LIN {X 0,Y 478.085,Z 266.813,A -85,B 0,C 180,E1 -7443.362,E2 -7443.362} C_VEL
LIN {X 0,Y 477.096,Z 286.447,A -85,B 0,C 180,E1 -7446.564,E2 -7446.564} C_VEL
LIN {X 0,Y 476.264,Z 303.664,A -85,B 0,C 180,E1 -7449.322,E2 -7449.322} C_VEL
LIN {X 0,Y 475.51,Z 306.267,A -85,B 0,C 180,E1 -7449.709,E2 -7449.709} C_VEL
LIN {X 0,Y 472.704,Z 310.776,A -85,B 0,C 180,E1 -7450.267,E2 -7450.267} C_VEL
LIN {X 0,Y 470.629,Z 314.949,A -85,B 0,C 180,E1 -7450.608,E2 -7450.608} C_VEL
LIN {X 0,Y 469.97,Z 318.585,A -85,B 0,C 180,E1 -7450.782,E2 -7450.782} C_VEL
LIN {X 0,Y 470.058,Z 319.87,A -85,B 0,C 180,E1 -7450.817,E2 -7450.817} C_VEL
LIN {X 0,Y 472.099,Z 332.179,A -85,B 0,C 180,E1 -7451.086,E2 -7451.086} C_VEL
LIN {X 0,Y 471.485,Z 425.613,A -85,B 0,C 180,E1 -7452.46,E2 -7452.46} C_VEL
LIN {X 0,Y 471.141,Z 438.708,A -85,B 0,C 180,E1 -7452.822,E2 -7452.822} C_VEL
LIN {X 0,Y 470.776,Z 451.277,A -85,B 0,C 180,E1 -7453.35,E2 -7453.35} C_VEL
LIN {X 0,Y 470.207,Z 463.7,A -85,B 0,C 180,E1 -7454.059,E2 -7454.059} C_VEL
LIN {X 0,Y 469.557,Z 475.266,A -85,B 0,C 180,E1 -7454.927,E2 -7454.927} C_VEL
LIN {X 0,Y 468.97,Z 485.65,A -85,B 0,C 180,E1 -7455.906,E2 -7455.906} C_VEL
LIN {X 0,Y 468.372,Z 495.014,A -85,B 0,C 180,E1 -7456.993,E2 -7456.993} C_VEL
LIN {X 0,Y 467.948,Z 502.687,A -85,B 0,C 180,E1 -7458.082,E2 -7458.082} C_VEL
LIN {X 0,Y 467.497,Z 510.197,A -85,B 0,C 180,E1 -7459.388,E2 -7459.388} C_VEL
LIN {X 0,Y 467.123,Z 517.124,A -85,B 0,C 180,E1 -7460.911,E2 -7460.911} C_VEL
LIN {X 0,Y 466.94,Z 521.744,A -85,B 0,C 180,E1 -7462.215,E2 -7462.215} C_VEL
LIN {X 0,Y 466.794,Z 525.41,A -85,B 0,C 180,E1 -7463.564,E2 -7463.564} C_VEL
LIN {X 0,Y 466.711,Z 527.879,A -85,B 0,C 180,E1 -7464.816,E2 -7464.816} C_VEL
LIN {X 0,Y 466.716,Z 529.948,A -85,B 0,C 180,E1 -7466.547,E2 -7466.547} C_VEL
LIN {X 0,Y 466.632,Z 530.463,A -85,B 0,C 180,E1 -7468.274,E2 -7468.274} C_VEL
LIN {X 0,Y 466.604,Z 529.509,A -85,B 0,C 180,E1 -7470,E2 -7470} C_VEL
LIN {X 0,Y 466.628,Z 528.478,A -85,B 0,C 180,E1 -7470.863,E2 -7470.863} C_VEL
LIN {X 0,Y 466.719,Z 527.02,A -85,B 0,C 180,E1 -7471.726,E2 -7471.726} C_VEL
LIN {X 0,Y 466.936,Z 522.899,A -85,B 0,C 180,E1 -7473.451,E2 -7473.451} C_VEL
LIN {X 0,Y 467.13,Z 518.624,A -85,B 0,C 180,E1 -7474.746,E2 -7474.746} C_VEL
LIN {X 0,Y 467.264,Z 513.213,A -85,B 0,C 180,E1 -7476.043,E2 -7476.043} C_VEL
LIN {X 0,Y 467.751,Z 506.1,A -85,B 0,C 180,E1 -7477.402,E2 -7477.402} C_VEL
LIN {X 0,Y 468.164,Z 498.071,A -85,B 0,C 180,E1 -7478.634,E2 -7478.634} C_VEL
LIN {X 0,Y 468.673,Z 489.478,A -85,B 0,C 180,E1 -7479.712,E2 -7479.712} C_VEL
LIN {X 0,Y 469.27,Z 478.914,A -85,B 0,C 180,E1 -7480.79,E2 -7480.79} C_VEL
LIN {X 0,Y 469.812,Z 468.39,A -85,B 0,C 180,E1 -7481.651,E2 -7481.651} C_VEL
LIN {X 0,Y 470.413,Z 456.63,A -85,B 0,C 180,E1 -7482.401,E2 -7482.401} C_VEL
LIN {X 0,Y 470.831,Z 444.4,A -85,B 0,C 180,E1 -7482.993,E2 -7482.993} C_VEL
LIN {X 0,Y 471.2,Z 431.794,A -85,B 0,C 180,E1 -7483.421,E2 -7483.421} C_VEL
LIN {X 0,Y 471.404,Z 418.703,A -85,B 0,C 180,E1 -7483.69,E2 -7483.69} C_VEL
LIN {X 0,Y 471.889,Z 331.972,A -85,B 0,C 180,E1 -7484.942,E2 -7484.942} C_VEL
LIN {X 0,Y 468.922,Z 314.095,A -85,B 0,C 180,E1 -7485.344,E2 -7485.344} C_VEL
LIN {X 0,Y 469.676,Z 295.344,A -85,B 0,C 180,E1 -7488.314,E2 -7488.314} C_VEL
LIN {X 0,Y 470.606,Z 276.031,A -85,B 0,C 180,E1 -7491.461,E2 -7491.461} C_VEL
LIN {X 0,Y 471.155,Z 266.374,A -85,B 0,C 180,E1 -7493.051,E2 -7493.051} C_VEL
LIN {X 0,Y 468.554,Z 254.185,A -85,B 0,C 180,E1 -7495.274,E2 -7495.274} C_VEL
LIN {X 0,Y 467.634,Z 249.988,A -85,B 0,C 180,E1 -7496.077,E2 -7496.077} C_VEL
LIN {X 0,Y 467.579,Z 249.864,A -85,B 0,C 180,E1 -7498.749,E2 -7498.749} C_VEL
LIN {X 0,Y 467.585,Z 249.866,A -85,B 0,C 180,E1 -7501.739,E2 -7501.739} C_VEL
LIN {X 0,Y 467.565,Z 249.859,A -85,B 0,C 180,E1 -7504.832,E2 -7504.832} C_VEL
LIN {X 0,Y 467.565,Z 249.864,A -85,B 0,C 180,E1 -7508.044,E2 -7508.044} C_VEL
LIN {X 0,Y 467.582,Z 249.863,A -85,B 0,C 180,E1 -7511.276,E2 -7511.276} C_VEL
LIN {X 0,Y 467.566,Z 249.864,A -85,B 0,C 180,E1 -7513.822,E2 -7513.822} C_VEL
LIN {X 0,Y 467.554,Z 249.863,A -85,B 0,C 180,E1 -7516.255,E2 -7516.255} C_VEL
LIN {X 0,Y 467.576,Z 249.866,A -85,B 0,C 180,E1 -7518.722,E2 -7518.722} C_VEL
LIN {X 0,Y 467.563,Z 249.864,A -85,B 0,C 180,E1 -7521.955,E2 -7521.955} C_VEL
LIN {X 0,Y 467.565,Z 249.858,A -85,B 0,C 180,E1 -7525.167,E2 -7525.167} C_VEL
LIN {X 0,Y 467.582,Z 249.859,A -85,B 0,C 180,E1 -7528.259,E2 -7528.259} C_VEL
LIN {X 0,Y 467.578,Z 249.863,A -85,B 0,C 180,E1 -7531.25,E2 -7531.25} C_VEL
LIN {X 0,Y 467.605,Z 249.86,A -85,B 0,C 180,E1 -7534.159,E2 -7534.159} C_VEL
LIN {X 0,Y 467.572,Z 249.87,A -85,B 0,C 180,E1 -7536.995,E2 -7536.995} C_VEL
LIN {X 0,Y 467.617,Z 249.854,A -85,B 0,C 180,E1 -7539.777,E2 -7539.777} C_VEL
LIN {X 0,Y 467.604,Z 249.863,A -85,B 0,C 180,E1 -7542.506,E2 -7542.506} C_VEL
LIN {X 0,Y 467.601,Z 249.859,A -85,B 0,C 180,E1 -7545.196,E2 -7545.196} C_VEL
LIN {X 0,Y 467.649,Z 249.854,A -85,B 0,C 180,E1 -7547.854,E2 -7547.854} C_VEL
LIN {X 0,Y 467.675,Z 249.85,A -85,B 0,C 180,E1 -7551.357,E2 -7551.357} C_VEL
LIN {X 0,Y 467.737,Z 249.844,A -85,B 0,C 180,E1 -7553.962,E2 -7553.962} C_VEL
LIN {X 0,Y 467.853,Z 249.828,A -85,B 0,C 180,E1 -7557.417,E2 -7557.417} C_VEL
LIN {X 0,Y 467.875,Z 249.826,A -85,B 0,C 180,E1 -7560,E2 -7560} C_VEL
LIN {X 0,Y 467.853,Z 249.834,A -85,B 0,C 180,E1 -7562.583,E2 -7562.583} C_VEL
LIN {X 0,Y 467.736,Z 249.842,A -85,B 0,C 180,E1 -7566.037,E2 -7566.037} C_VEL
LIN {X 0,Y 467.674,Z 249.854,A -85,B 0,C 180,E1 -7568.643,E2 -7568.643} C_VEL
LIN {X 0,Y 467.648,Z 249.855,A -85,B 0,C 180,E1 -7572.145,E2 -7572.145} C_VEL
LIN {X 0,Y 467.632,Z 249.855,A -85,B 0,C 180,E1 -7575.695,E2 -7575.695} C_VEL
LIN {X 0,Y 467.61,Z 249.859,A -85,B 0,C 180,E1 -7578.765,E2 -7578.765} C_VEL
LIN {X 0,Y 467.573,Z 249.861,A -85,B 0,C 180,E1 -7581.268,E2 -7581.268} C_VEL
LIN {X 0,Y 467.567,Z 249.869,A -85,B 0,C 180,E1 -7583.943,E2 -7583.943} C_VEL
LIN {X 0,Y 467.61,Z 249.859,A -85,B 0,C 180,E1 -7586.801,E2 -7586.801} C_VEL
LIN {X 0,Y 467.581,Z 249.856,A -85,B 0,C 180,E1 -7589.736,E2 -7589.736} C_VEL
LIN {X 0,Y 467.578,Z 249.863,A -85,B 0,C 180,E1 -7592.759,E2 -7592.759} C_VEL
LIN {X 0,Y 467.551,Z 249.863,A -85,B 0,C 180,E1 -7595.89,E2 -7595.89} C_VEL
LIN {X 0,Y 467.577,Z 249.864,A -85,B 0,C 180,E1 -7599.145,E2 -7599.145} C_VEL
LIN {X 0,Y 467.582,Z 249.859,A -85,B 0,C 180,E1 -7602.567,E2 -7602.567} C_VEL
LIN {X 0,Y 467.566,Z 249.866,A -85,B 0,C 180,E1 -7605.054,E2 -7605.054} C_VEL
LIN {X 0,Y 467.585,Z 249.844,A -85,B 0,C 180,E1 -7607.44,E2 -7607.44} C_VEL
LIN {X 0,Y 467.578,Z 249.863,A -85,B 0,C 180,E1 -7610.856,E2 -7610.856} C_VEL
LIN {X 0,Y 467.557,Z 249.852,A -85,B 0,C 180,E1 -7614.261,E2 -7614.261} C_VEL
LIN {X 0,Y 467.58,Z 249.861,A -85,B 0,C 180,E1 -7617.321,E2 -7617.321} C_VEL
LIN {X 0,Y 467.568,Z 249.865,A -85,B 0,C 180,E1 -7620.668,E2 -7620.668} C_VEL
LIN {X 0,Y 467.679,Z 249.999,A -85,B 0,C 180,E1 -7622.625,E2 -7622.625} C_VEL
LIN {X 0,Y 471.47,Z 266.255,A -85,B 0,C 180,E1 -7625.331,E2 -7625.331} C_VEL
LIN {X 0,Y 471.671,Z 269.572,A -85,B 0,C 180,E1 -7625.836,E2 -7625.836} C_VEL
LIN {X 0,Y 470.357,Z 291.394,A -85,B 0,C 180,E1 -7628.986,E2 -7628.986} C_VEL
LIN {X 0,Y 470.145,Z 296.887,A -85,B 0,C 180,E1 -7629.737,E2 -7629.737} C_VEL
LIN {X 0,Y 472.697,Z 313.021,A -85,B 0,C 180,E1 -7630.12,E2 -7630.12} C_VEL
LIN {X 0,Y 471.417,Z 431.926,A -85,B 0,C 180,E1 -7632.037,E2 -7632.037} C_VEL
LIN {X 0,Y 471.033,Z 446.54,A -85,B 0,C 180,E1 -7632.442,E2 -7632.442} C_VEL
LIN {X 0,Y 470.559,Z 460.601,A -85,B 0,C 180,E1 -7633.016,E2 -7633.016} C_VEL
LIN {X 0,Y 470.028,Z 473.558,A -85,B 0,C 180,E1 -7633.719,E2 -7633.719} C_VEL
LIN {X 0,Y 469.39,Z 486.203,A -85,B 0,C 180,E1 -7634.588,E2 -7634.588} C_VEL
LIN {X 0,Y 468.797,Z 497.744,A -85,B 0,C 180,E1 -7635.568,E2 -7635.568} C_VEL
LIN {X 0,Y 468.358,Z 507.345,A -85,B 0,C 180,E1 -7636.551,E2 -7636.551} C_VEL
LIN {X 0,Y 467.91,Z 518.036,A -85,B 0,C 180,E1 -7637.862,E2 -7637.862} C_VEL
LIN {X 0,Y 467.454,Z 526.834,A -85,B 0,C 180,E1 -7639.168,E2 -7639.168} C_VEL
LIN {X 0,Y 467.105,Z 535.228,A -85,B 0,C 180,E1 -7640.692,E2 -7640.692} C_VEL
LIN {X 0,Y 466.851,Z 541.954,A -85,B 0,C 180,E1 -7642.213,E2 -7642.213} C_VEL
LIN {X 0,Y 466.757,Z 546.875,A -85,B 0,C 180,E1 -7643.6,E2 -7643.6} C_VEL
LIN {X 0,Y 466.723,Z 550.262,A -85,B 0,C 180,E1 -7644.816,E2 -7644.816} C_VEL
LIN {X 0,Y 466.679,Z 553.826,A -85,B 0,C 180,E1 -7646.547,E2 -7646.547} C_VEL
LIN {X 0,Y 466.604,Z 555.941,A -85,B 0,C 180,E1 -7648.274,E2 -7648.274} C_VEL
LIN {X 0,Y 466.597,Z 556.653,A -85,B 0,C 180,E1 -7650,E2 -7650} C_VEL
LIN {X 0,Y 466.604,Z 555.958,A -85,B 0,C 180,E1 -7651.726,E2 -7651.726} C_VEL
LIN {X 0,Y 466.679,Z 553.86,A -85,B 0,C 180,E1 -7653.453,E2 -7653.453} C_VEL
LIN {X 0,Y 466.727,Z 550.313,A -85,B 0,C 180,E1 -7655.184,E2 -7655.184} C_VEL
LIN {X 0,Y 466.82,Z 545.216,A -85,B 0,C 180,E1 -7656.917,E2 -7656.917} C_VEL
LIN {X 0,Y 466.947,Z 540.274,A -85,B 0,C 180,E1 -7658.22,E2 -7658.22} C_VEL
LIN {X 0,Y 467.177,Z 533.133,A -85,B 0,C 180,E1 -7659.743,E2 -7659.743} C_VEL
LIN {X 0,Y 467.617,Z 524.274,A -85,B 0,C 180,E1 -7661.267,E2 -7661.267} C_VEL
LIN {X 0,Y 468.088,Z 514.113,A -85,B 0,C 180,E1 -7662.69,E2 -7662.69} C_VEL
LIN {X 0,Y 468.575,Z 503.701,A -85,B 0,C 180,E1 -7663.885,E2 -7663.885} C_VEL
LIN {X 0,Y 469.161,Z 492.153,A -85,B 0,C 180,E1 -7664.975,E2 -7664.975} C_VEL
LIN {X 0,Y 469.84,Z 479.364,A -85,B 0,C 180,E1 -7665.953,E2 -7665.953} C_VEL
LIN {X 0,Y 470.412,Z 465.977,A -85,B 0,C 180,E1 -7666.766,E2 -7666.766} C_VEL
LIN {X 0,Y 470.96,Z 451.819,A -85,B 0,C 180,E1 -7667.42,E2 -7667.42} C_VEL
LIN {X 0,Y 471.441,Z 437.698,A -85,B 0,C 180,E1 -7667.878,E2 -7667.878} C_VEL
LIN {X 0,Y 471.723,Z 421.368,A -85,B 0,C 180,E1 -7668.204,E2 -7668.204} C_VEL
LIN {X 0,Y 472.823,Z 312.677,A -85,B 0,C 180,E1 -7669.954,E2 -7669.954} C_VEL
LIN {X 0,Y 470.225,Z 296.843,A -85,B 0,C 180,E1 -7670.346,E2 -7670.346} C_VEL
LIN {X 0,Y 471.398,Z 276.465,A -85,B 0,C 180,E1 -7673.271,E2 -7673.271} C_VEL
LIN {X 0,Y 471.885,Z 268.33,A -85,B 0,C 180,E1 -7674.461,E2 -7674.461} C_VEL
LIN {X 0,Y 468.859,Z 254.709,A -85,B 0,C 180,E1 -7676.723,E2 -7676.723} C_VEL
LIN {X 0,Y 467.644,Z 249.964,A -85,B 0,C 180,E1 -7677.581,E2 -7677.581} C_VEL
LIN {X 0,Y 467.567,Z 249.86,A -85,B 0,C 180,E1 -7681.045,E2 -7681.045} C_VEL
LIN {X 0,Y 467.586,Z 249.869,A -85,B 0,C 180,E1 -7684.242,E2 -7684.242} C_VEL
LIN {X 0,Y 467.545,Z 249.857,A -85,B 0,C 180,E1 -7687.186,E2 -7687.186} C_VEL
LIN {X 0,Y 467.575,Z 249.865,A -85,B 0,C 180,E1 -7690.264,E2 -7690.264} C_VEL
LIN {X 0,Y 467.616,Z 249.863,A -85,B 0,C 180,E1 -7692.571,E2 -7692.571} C_VEL
LIN {X 0,Y 467.567,Z 249.862,A -85,B 0,C 180,E1 -7695.053,E2 -7695.053} C_VEL
LIN {X 0,Y 467.585,Z 249.862,A -85,B 0,C 180,E1 -7697.44,E2 -7697.44} C_VEL
LIN {X 0,Y 467.578,Z 249.865,A -85,B 0,C 180,E1 -7700.855,E2 -7700.855} C_VEL
LIN {X 0,Y 467.558,Z 249.86,A -85,B 0,C 180,E1 -7704.26,E2 -7704.26} C_VEL
LIN {X 0,Y 467.577,Z 249.864,A -85,B 0,C 180,E1 -7707.32,E2 -7707.32} C_VEL
LIN {X 0,Y 467.571,Z 249.855,A -85,B 0,C 180,E1 -7710.666,E2 -7710.666} C_VEL
LIN {X 0,Y 467.61,Z 249.859,A -85,B 0,C 180,E1 -7713.199,E2 -7713.199} C_VEL
LIN {X 0,Y 467.587,Z 249.863,A -85,B 0,C 180,E1 -7716.468,E2 -7716.468} C_VEL
LIN {X 0,Y 467.616,Z 249.86,A -85,B 0,C 180,E1 -7719.777,E2 -7719.777} C_VEL
LIN {X 0,Y 467.603,Z 249.859,A -85,B 0,C 180,E1 -7722.507,E2 -7722.507} C_VEL
LIN {X 0,Y 467.6,Z 249.86,A -85,B 0,C 180,E1 -7725.196,E2 -7725.196} C_VEL
LIN {X 0,Y 467.649,Z 249.854,A -85,B 0,C 180,E1 -7727.855,E2 -7727.855} C_VEL
LIN {X 0,Y 467.675,Z 249.854,A -85,B 0,C 180,E1 -7731.357,E2 -7731.357} C_VEL
LIN {X 0,Y 467.737,Z 249.847,A -85,B 0,C 180,E1 -7733.963,E2 -7733.963} C_VEL
LIN {X 0,Y 467.853,Z 249.83,A -85,B 0,C 180,E1 -7737.417,E2 -7737.417} C_VEL
LIN {X 0,Y 467.876,Z 249.828,A -85,B 0,C 180,E1 -7740,E2 -7740} C_VEL
LIN {X 0,Y 467.854,Z 249.823,A -85,B 0,C 180,E1 -7742.583,E2 -7742.583} C_VEL
LIN {X 0,Y 467.737,Z 249.841,A -85,B 0,C 180,E1 -7746.038,E2 -7746.038} C_VEL
LIN {X 0,Y 467.676,Z 249.85,A -85,B 0,C 180,E1 -7748.643,E2 -7748.643} C_VEL
LIN {X 0,Y 467.65,Z 249.852,A -85,B 0,C 180,E1 -7752.146,E2 -7752.146} C_VEL
LIN {X 0,Y 467.633,Z 249.855,A -85,B 0,C 180,E1 -7755.696,E2 -7755.696} C_VEL
LIN {X 0,Y 467.612,Z 249.861,A -85,B 0,C 180,E1 -7758.765,E2 -7758.765} C_VEL
LIN {X 0,Y 467.576,Z 249.869,A -85,B 0,C 180,E1 -7761.269,E2 -7761.269} C_VEL
LIN {X 0,Y 467.568,Z 249.862,A -85,B 0,C 180,E1 -7763.944,E2 -7763.944} C_VEL
LIN {X 0,Y 467.613,Z 249.863,A -85,B 0,C 180,E1 -7766.801,E2 -7766.801} C_VEL
LIN {X 0,Y 467.55,Z 249.861,A -85,B 0,C 180,E1 -7769.739,E2 -7769.739} C_VEL
LIN {X 0,Y 467.581,Z 249.868,A -85,B 0,C 180,E1 -7772.759,E2 -7772.759} C_VEL
LIN {X 0,Y 467.554,Z 249.861,A -85,B 0,C 180,E1 -7775.89,E2 -7775.89} C_VEL
LIN {X 0,Y 467.574,Z 249.86,A -85,B 0,C 180,E1 -7779.146,E2 -7779.146} C_VEL
LIN {X 0,Y 467.585,Z 249.867,A -85,B 0,C 180,E1 -7782.568,E2 -7782.568} C_VEL
LIN {X 0,Y 467.57,Z 249.868,A -85,B 0,C 180,E1 -7785.054,E2 -7785.054} C_VEL
LIN {X 0,Y 467.589,Z 249.859,A -85,B 0,C 180,E1 -7787.441,E2 -7787.441} C_VEL
LIN {X 0,Y 467.582,Z 249.851,A -85,B 0,C 180,E1 -7790.856,E2 -7790.856} C_VEL
LIN {X 0,Y 467.56,Z 249.871,A -85,B 0,C 180,E1 -7794.262,E2 -7794.262} C_VEL
LIN {X 0,Y 467.581,Z 249.867,A -85,B 0,C 180,E1 -7797.322,E2 -7797.322} C_VEL
LIN {X 0,Y 467.596,Z 250.065,A -85,B 0,C 180,E1 -7799.831,E2 -7799.831} C_VEL
LIN {X 0,Y 470.568,Z 262.803,A -85,B 0,C 180,E1 -7802.246,E2 -7802.246} C_VEL
LIN {X 0,Y 471.257,Z 268.059,A -85,B 0,C 180,E1 -7803.184,E2 -7803.184} C_VEL
LIN {X 0,Y 470.191,Z 287.705,A -85,B 0,C 180,E1 -7806.433,E2 -7806.433} C_VEL
LIN {X 0,Y 469.158,Z 308.757,A -85,B 0,C 180,E1 -7809.847,E2 -7809.847} C_VEL
LIN {X 0,Y 469.023,Z 313.903,A -85,B 0,C 180,E1 -7810.648,E2 -7810.648} C_VEL
LIN {X 0,Y 470.058,Z 319.87,A -85,B 0,C 180,E1 -7810.817,E2 -7810.817} C_VEL
LIN {X 0,Y 470.179,Z 325.726,A -85,B 0,C 180,E1 -7810.91,E2 -7810.91} C_VEL
LIN {X 0,Y 469.247,Z 331.594,A -85,B 0,C 180,E1 -7810.958,E2 -7810.958} C_VEL
LIN {X 0,Y 466.333,Z 343.281,A -85,B 0,C 180,E1 -7811.009,E2 -7811.009} C_VEL
LIN {X 0,Y 465.398,Z 349.209,A -85,B 0,C 180,E1 -7811.058,E2 -7811.058} C_VEL
LIN {X 0,Y 465.298,Z 351.201,A -85,B 0,C 180,E1 -7811.084,E2 -7811.084} C_VEL
LIN {X 0,Y 464.726,Z 425.765,A -85,B 0,C 180,E1 -7812.196,E2 -7812.196} C_VEL
LIN {X 0,Y 464.36,Z 439.005,A -85,B 0,C 180,E1 -7812.569,E2 -7812.569} C_VEL
LIN {X 0,Y 463.967,Z 451.581,A -85,B 0,C 180,E1 -7813.107,E2 -7813.107} C_VEL
LIN {X 0,Y 463.395,Z 463.826,A -85,B 0,C 180,E1 -7813.819,E2 -7813.819} C_VEL
LIN {X 0,Y 462.694,Z 475.393,A -85,B 0,C 180,E1 -7814.698,E2 -7814.698} C_VEL
LIN {X 0,Y 462.066,Z 485.78,A -85,B 0,C 180,E1 -7815.691,E2 -7815.691} C_VEL
LIN {X 0,Y 461.419,Z 495.148,A -85,B 0,C 180,E1 -7816.793,E2 -7816.793} C_VEL
LIN {X 0,Y 460.977,Z 502.825,A -85,B 0,C 180,E1 -7817.899,E2 -7817.899} C_VEL
LIN {X 0,Y 460.498,Z 510.341,A -85,B 0,C 180,E1 -7819.225,E2 -7819.225} C_VEL
LIN {X 0,Y 460.093,Z 517.272,A -85,B 0,C 180,E1 -7820.771,E2 -7820.771} C_VEL
LIN {X 0,Y 459.886,Z 521.898,A -85,B 0,C 180,E1 -7822.095,E2 -7822.095} C_VEL
LIN {X 0,Y 459.717,Z 525.817,A -85,B 0,C 180,E1 -7823.569,E2 -7823.569} C_VEL
LIN {X 0,Y 459.646,Z 528.049,A -85,B 0,C 180,E1 -7824.736,E2 -7824.736} C_VEL
LIN {X 0,Y 459.613,Z 530.13,A -85,B 0,C 180,E1 -7826.493,E2 -7826.493} C_VEL
LIN {X 0,Y 459.585,Z 530.591,A -85,B 0,C 180,E1 -7827.371,E2 -7827.371} C_VEL
LIN {X 0,Y 459.525,Z 530.378,A -85,B 0,C 180,E1 -7829.124,E2 -7829.124} C_VEL
LIN {X 0,Y 459.562,Z 528.711,A -85,B 0,C 180,E1 -7830.876,E2 -7830.876} C_VEL
LIN {X 0,Y 459.627,Z 527.272,A -85,B 0,C 180,E1 -7831.752,E2 -7831.752} C_VEL
LIN {X 0,Y 459.867,Z 523.177,A -85,B 0,C 180,E1 -7833.505,E2 -7833.505} C_VEL
LIN {X 0,Y 460.069,Z 518.929,A -85,B 0,C 180,E1 -7834.819,E2 -7834.819} C_VEL
LIN {X 0,Y 460.291,Z 512.552,A -85,B 0,C 180,E1 -7836.355,E2 -7836.355} C_VEL
LIN {X 0,Y 460.777,Z 505.573,A -85,B 0,C 180,E1 -7837.669,E2 -7837.669} C_VEL
LIN {X 0,Y 461.172,Z 498.514,A -85,B 0,C 180,E1 -7838.765,E2 -7838.765} C_VEL
LIN {X 0,Y 461.703,Z 489.98,A -85,B 0,C 180,E1 -7839.86,E2 -7839.86} C_VEL
LIN {X 0,Y 462.332,Z 479.485,A -85,B 0,C 180,E1 -7840.953,E2 -7840.953} C_VEL
LIN {X 0,Y 462.909,Z 469.056,A -85,B 0,C 180,E1 -7841.827,E2 -7841.827} C_VEL
LIN {X 0,Y 463.545,Z 457.506,A -85,B 0,C 180,E1 -7842.588,E2 -7842.588} C_VEL
LIN {X 0,Y 463.965,Z 445.517,A -85,B 0,C 180,E1 -7843.189,E2 -7843.189} C_VEL
LIN {X 0,Y 464.384,Z 432.407,A -85,B 0,C 180,E1 -7843.65,E2 -7843.65} C_VEL
LIN {X 0,Y 464.611,Z 419.813,A -85,B 0,C 180,E1 -7843.922,E2 -7843.922} C_VEL
LIN {X 0,Y 465.011,Z 331.821,A -85,B 0,C 180,E1 -7845.213,E2 -7845.213} C_VEL
LIN {X 0,Y 462.025,Z 314.35,A -85,B 0,C 180,E1 -7845.607,E2 -7845.607} C_VEL
LIN {X 0,Y 461.99,Z 313.56,A -85,B 0,C 180,E1 -7845.665,E2 -7845.665} C_VEL
LIN {X 0,Y 462.925,Z 292.706,A -85,B 0,C 180,E1 -7849.05,E2 -7849.05} C_VEL
LIN {X 0,Y 463.914,Z 273.38,A -85,B 0,C 180,E1 -7852.255,E2 -7852.255} C_VEL
LIN {X 0,Y 464.285,Z 267.857,A -85,B 0,C 180,E1 -7853.176,E2 -7853.176} C_VEL
LIN {X 0,Y 461.309,Z 254.051,A -85,B 0,C 180,E1 -7855.741,E2 -7855.741} C_VEL
LIN {X 0,Y 460.582,Z 250.828,A -85,B 0,C 180,E1 -7856.385,E2 -7856.385} C_VEL
LIN {X 0,Y 460.542,Z 250.734,A -85,B 0,C 180,E1 -7859.23,E2 -7859.23} C_VEL
LIN {X 0,Y 460.533,Z 250.741,A -85,B 0,C 180,E1 -7862.284,E2 -7862.284} C_VEL
LIN {X 0,Y 460.511,Z 250.745,A -85,B 0,C 180,E1 -7865.445,E2 -7865.445} C_VEL
LIN {X 0,Y 460.544,Z 250.741,A -85,B 0,C 180,E1 -7868.897,E2 -7868.897} C_VEL
LIN {X 0,Y 460.523,Z 250.742,A -85,B 0,C 180,E1 -7872.18,E2 -7872.18} C_VEL
LIN {X 0,Y 460.516,Z 250.741,A -85,B 0,C 180,E1 -7875.411,E2 -7875.411} C_VEL
LIN {X 0,Y 460.53,Z 250.741,A -85,B 0,C 180,E1 -7878.397,E2 -7878.397} C_VEL
LIN {X 0,Y 460.517,Z 250.741,A -85,B 0,C 180,E1 -7881.265,E2 -7881.265} C_VEL
LIN {X 0,Y 460.51,Z 250.744,A -85,B 0,C 180,E1 -7884.554,E2 -7884.554} C_VEL
LIN {X 0,Y 460.529,Z 250.737,A -85,B 0,C 180,E1 -7887.715,E2 -7887.715} C_VEL
LIN {X 0,Y 460.543,Z 250.745,A -85,B 0,C 180,E1 -7890.769,E2 -7890.769} C_VEL
LIN {X 0,Y 460.558,Z 250.738,A -85,B 0,C 180,E1 -7893.734,E2 -7893.734} C_VEL
LIN {X 0,Y 460.541,Z 250.739,A -85,B 0,C 180,E1 -7896.623,E2 -7896.623} C_VEL
LIN {X 0,Y 460.545,Z 250.736,A -85,B 0,C 180,E1 -7899.452,E2 -7899.452} C_VEL
LIN {X 0,Y 460.554,Z 250.739,A -85,B 0,C 180,E1 -7902.23,E2 -7902.23} C_VEL
LIN {X 0,Y 460.559,Z 250.737,A -85,B 0,C 180,E1 -7904.964,E2 -7904.964} C_VEL
LIN {X 0,Y 460.602,Z 250.732,A -85,B 0,C 180,E1 -7907.665,E2 -7907.665} C_VEL
LIN {X 0,Y 460.622,Z 250.729,A -85,B 0,C 180,E1 -7911.223,E2 -7911.223} C_VEL
LIN {X 0,Y 460.703,Z 250.719,A -85,B 0,C 180,E1 -7913.87,E2 -7913.87} C_VEL
LIN {X 0,Y 460.818,Z 250.705,A -85,B 0,C 180,E1 -7917.377,E2 -7917.377} C_VEL
LIN {X 0,Y 460.846,Z 250.702,A -85,B 0,C 180,E1 -7920,E2 -7920} C_VEL
LIN {X 0,Y 460.818,Z 250.71,A -85,B 0,C 180,E1 -7922.622,E2 -7922.622} C_VEL
LIN {X 0,Y 460.703,Z 250.718,A -85,B 0,C 180,E1 -7926.13,E2 -7926.13} C_VEL
LIN {X 0,Y 460.622,Z 250.731,A -85,B 0,C 180,E1 -7928.776,E2 -7928.776} C_VEL
LIN {X 0,Y 460.606,Z 250.737,A -85,B 0,C 180,E1 -7932.445,E2 -7932.445} C_VEL
LIN {X 0,Y 460.593,Z 250.733,A -85,B 0,C 180,E1 -7935.998,E2 -7935.998} C_VEL
LIN {X 0,Y 460.563,Z 250.736,A -85,B 0,C 180,E1 -7938.902,E2 -7938.902} C_VEL
LIN {X 0,Y 460.509,Z 250.742,A -85,B 0,C 180,E1 -7941.486,E2 -7941.486} C_VEL
LIN {X 0,Y 460.536,Z 250.74,A -85,B 0,C 180,E1 -7944.332,E2 -7944.332} C_VEL
LIN {X 0,Y 460.573,Z 250.736,A -85,B 0,C 180,E1 -7947.244,E2 -7947.244} C_VEL
LIN {X 0,Y 460.521,Z 250.731,A -85,B 0,C 180,E1 -7950.239,E2 -7950.239} C_VEL
LIN {X 0,Y 460.524,Z 250.743,A -85,B 0,C 180,E1 -7953.325,E2 -7953.325} C_VEL
LIN {X 0,Y 460.473,Z 250.737,A -85,B 0,C 180,E1 -7956.53,E2 -7956.53} C_VEL
LIN {X 0,Y 460.553,Z 250.745,A -85,B 0,C 180,E1 -7959.86,E2 -7959.86} C_VEL
LIN {X 0,Y 460.508,Z 250.74,A -85,B 0,C 180,E1 -7962.901,E2 -7962.901} C_VEL
LIN {X 0,Y 460.505,Z 250.74,A -85,B 0,C 180,E1 -7965.831,E2 -7965.831} C_VEL
LIN {X 0,Y 460.527,Z 250.722,A -85,B 0,C 180,E1 -7968.989,E2 -7968.989} C_VEL
LIN {X 0,Y 460.522,Z 250.746,A -85,B 0,C 180,E1 -7971.267,E2 -7971.267} C_VEL
LIN {X 0,Y 460.507,Z 250.73,A -85,B 0,C 180,E1 -7974.555,E2 -7974.555} C_VEL
LIN {X 0,Y 460.529,Z 250.733,A -85,B 0,C 180,E1 -7977.716,E2 -7977.716} C_VEL
LIN {X 0,Y 460.538,Z 250.738,A -85,B 0,C 180,E1 -7980.77,E2 -7980.77} C_VEL
LIN {X 0,Y 460.646,Z 250.959,A -85,B 0,C 180,E1 -7982.341,E2 -7982.341} C_VEL
LIN {X 0,Y 464.19,Z 266.18,A -85,B 0,C 180,E1 -7984.918,E2 -7984.918} C_VEL
LIN {X 0,Y 464.86,Z 270.105,A -85,B 0,C 180,E1 -7985.55,E2 -7985.55} C_VEL
LIN {X 0,Y 463.651,Z 289.726,A -85,B 0,C 180,E1 -7988.434,E2 -7988.434} C_VEL
LIN {X 0,Y 463.272,Z 297.079,A -85,B 0,C 180,E1 -7989.461,E2 -7989.461} C_VEL
LIN {X 0,Y 465.969,Z 313.961,A -85,B 0,C 180,E1 -7989.869,E2 -7989.869} C_VEL
LIN {X 0,Y 464.586,Z 432.822,A -85,B 0,C 180,E1 -7991.82,E2 -7991.82} C_VEL
LIN {X 0,Y 464.162,Z 447.086,A -85,B 0,C 180,E1 -7992.231,E2 -7992.231} C_VEL
LIN {X 0,Y 463.666,Z 460.989,A -85,B 0,C 180,E1 -7992.813,E2 -7992.813} C_VEL
LIN {X 0,Y 463.095,Z 474.719,A -85,B 0,C 180,E1 -7993.582,E2 -7993.582} C_VEL
LIN {X 0,Y 462.414,Z 487.118,A -85,B 0,C 180,E1 -7994.463,E2 -7994.463} C_VEL
LIN {X 0,Y 461.792,Z 498.474,A -85,B 0,C 180,E1 -7995.457,E2 -7995.457} C_VEL
LIN {X 0,Y 461.295,Z 508.92,A -85,B 0,C 180,E1 -7996.565,E2 -7996.565} C_VEL
LIN {X 0,Y 460.816,Z 519.265,A -85,B 0,C 180,E1 -7997.895,E2 -7997.895} C_VEL
LIN {X 0,Y 460.371,Z 527.818,A -85,B 0,C 180,E1 -7999.222,E2 -7999.222} C_VEL
LIN {X 0,Y 460.021,Z 535.972,A -85,B 0,C 180,E1 -8000.769,E2 -8000.769} C_VEL
LIN {X 0,Y 459.794,Z 541.69,A -85,B 0,C 180,E1 -8002.093,E2 -8002.093} C_VEL
LIN {X 0,Y 459.652,Z 547.023,A -85,B 0,C 180,E1 -8003.636,E2 -8003.636} C_VEL
LIN {X 0,Y 459.631,Z 550.027,A -85,B 0,C 180,E1 -8004.736,E2 -8004.736} C_VEL
LIN {X 0,Y 459.574,Z 553.606,A -85,B 0,C 180,E1 -8006.493,E2 -8006.493} C_VEL
LIN {X 0,Y 459.517,Z 555.733,A -85,B 0,C 180,E1 -8008.247,E2 -8008.247} C_VEL
LIN {X 0,Y 459.528,Z 556.454,A -85,B 0,C 180,E1 -8010,E2 -8010} C_VEL
LIN {X 0,Y 459.517,Z 555.764,A -85,B 0,C 180,E1 -8011.753,E2 -8011.753} C_VEL
LIN {X 0,Y 459.574,Z 553.666,A -85,B 0,C 180,E1 -8013.507,E2 -8013.507} C_VEL
LIN {X 0,Y 459.636,Z 550.116,A -85,B 0,C 180,E1 -8015.264,E2 -8015.264} C_VEL
LIN {X 0,Y 459.731,Z 545.014,A -85,B 0,C 180,E1 -8017.025,E2 -8017.025} C_VEL
LIN {X 0,Y 459.893,Z 540.068,A -85,B 0,C 180,E1 -8018.347,E2 -8018.347} C_VEL
LIN {X 0,Y 460.132,Z 532.918,A -85,B 0,C 180,E1 -8019.894,E2 -8019.894} C_VEL
LIN {X 0,Y 460.597,Z 524.051,A -85,B 0,C 180,E1 -8021.441,E2 -8021.441} C_VEL
LIN {X 0,Y 461.096,Z 514.261,A -85,B 0,C 180,E1 -8022.836,E2 -8022.836} C_VEL
LIN {X 0,Y 461.633,Z 503.447,A -85,B 0,C 180,E1 -8024.098,E2 -8024.098} C_VEL
LIN {X 0,Y 462.272,Z 491.882,A -85,B 0,C 180,E1 -8025.204,E2 -8025.204} C_VEL
LIN {X 0,Y 462.978,Z 479.067,A -85,B 0,C 180,E1 -8026.196,E2 -8026.196} C_VEL
LIN {X 0,Y 463.559,Z 466.214,A -85,B 0,C 180,E1 -8026.989,E2 -8026.989} C_VEL
LIN {X 0,Y 464.104,Z 452.72,A -85,B 0,C 180,E1 -8027.629,E2 -8027.629} C_VEL
LIN {X 0,Y 464.643,Z 438.198,A -85,B 0,C 180,E1 -8028.12,E2 -8028.12} C_VEL
LIN {X 0,Y 464.948,Z 422.205,A -85,B 0,C 180,E1 -8028.45,E2 -8028.45} C_VEL
LIN {X 0,Y 466.137,Z 313.522,A -85,B 0,C 180,E1 -8030.227,E2 -8030.227} C_VEL
LIN {X 0,Y 463.385,Z 296.925,A -85,B 0,C 180,E1 -8030.65,E2 -8030.65} C_VEL
LIN {X 0,Y 464.669,Z 276.542,A -85,B 0,C 180,E1 -8033.628,E2 -8033.628} C_VEL
LIN {X 0,Y 465.021,Z 269.577,A -85,B 0,C 180,E1 -8034.669,E2 -8034.669} C_VEL
LIN {X 0,Y 461.633,Z 254.823,A -85,B 0,C 180,E1 -8037.176,E2 -8037.176} C_VEL
LIN {X 0,Y 460.586,Z 250.85,A -85,B 0,C 180,E1 -8037.911,E2 -8037.911} C_VEL
LIN {X 0,Y 460.519,Z 250.734,A -85,B 0,C 180,E1 -8041.283,E2 -8041.283} C_VEL
LIN {X 0,Y 460.53,Z 250.744,A -85,B 0,C 180,E1 -8044.505,E2 -8044.505} C_VEL
LIN {X 0,Y 460.498,Z 250.737,A -85,B 0,C 180,E1 -8047.623,E2 -8047.623} C_VEL
LIN {X 0,Y 460.539,Z 250.741,A -85,B 0,C 180,E1 -8050.269,E2 -8050.269} C_VEL
LIN {X 0,Y 460.521,Z 250.742,A -85,B 0,C 180,E1 -8053.372,E2 -8053.372} C_VEL
LIN {X 0,Y 460.496,Z 250.748,A -85,B 0,C 180,E1 -8056.624,E2 -8056.624} C_VEL
LIN {X 0,Y 460.537,Z 250.736,A -85,B 0,C 180,E1 -8059.73,E2 -8059.73} C_VEL
LIN {X 0,Y 460.522,Z 250.739,A -85,B 0,C 180,E1 -8062.519,E2 -8062.519} C_VEL
LIN {X 0,Y 460.543,Z 250.737,A -85,B 0,C 180,E1 -8065.624,E2 -8065.624} C_VEL
LIN {X 0,Y 460.531,Z 250.735,A -85,B 0,C 180,E1 -8068.744,E2 -8068.744} C_VEL
LIN {X 0,Y 460.552,Z 250.733,A -85,B 0,C 180,E1 -8071.767,E2 -8071.767} C_VEL
LIN {X 0,Y 460.553,Z 250.737,A -85,B 0,C 180,E1 -8074.705,E2 -8074.705} C_VEL
LIN {X 0,Y 460.506,Z 250.747,A -85,B 0,C 180,E1 -8077.571,E2 -8077.571} C_VEL
LIN {X 0,Y 460.562,Z 250.738,A -85,B 0,C 180,E1 -8080.384,E2 -8080.384} C_VEL
LIN {X 0,Y 460.559,Z 250.736,A -85,B 0,C 180,E1 -8083.146,E2 -8083.146} C_VEL
LIN {X 0,Y 460.549,Z 250.744,A -85,B 0,C 180,E1 -8085.868,E2 -8085.868} C_VEL
LIN {X 0,Y 460.604,Z 250.728,A -85,B 0,C 180,E1 -8088.559,E2 -8088.559} C_VEL
LIN {X 0,Y 460.688,Z 250.718,A -85,B 0,C 180,E1 -8092.109,E2 -8092.109} C_VEL
LIN {X 0,Y 460.691,Z 250.721,A -85,B 0,C 180,E1 -8094.749,E2 -8094.749} C_VEL
LIN {X 0,Y 460.818,Z 250.706,A -85,B 0,C 180,E1 -8097.378,E2 -8097.378} C_VEL
LIN {X 0,Y 460.846,Z 250.703,A -85,B 0,C 180,E1 -8100,E2 -8100} C_VEL
LIN {X 0,Y 460.819,Z 250.7,A -85,B 0,C 180,E1 -8102.623,E2 -8102.623} C_VEL
LIN {X 0,Y 460.703,Z 250.716,A -85,B 0,C 180,E1 -8106.13,E2 -8106.13} C_VEL
LIN {X 0,Y 460.623,Z 250.729,A -85,B 0,C 180,E1 -8108.777,E2 -8108.777} C_VEL
LIN {X 0,Y 460.608,Z 250.729,A -85,B 0,C 180,E1 -8112.445,E2 -8112.445} C_VEL
LIN {X 0,Y 460.595,Z 250.73,A -85,B 0,C 180,E1 -8115.998,E2 -8115.998} C_VEL
LIN {X 0,Y 460.566,Z 250.74,A -85,B 0,C 180,E1 -8118.902,E2 -8118.902} C_VEL
LIN {X 0,Y 460.511,Z 250.748,A -85,B 0,C 180,E1 -8121.486,E2 -8121.486} C_VEL
LIN {X 0,Y 460.538,Z 250.738,A -85,B 0,C 180,E1 -8124.333,E2 -8124.333} C_VEL
LIN {X 0,Y 460.569,Z 250.734,A -85,B 0,C 180,E1 -8127.245,E2 -8127.245} C_VEL
LIN {X 0,Y 460.507,Z 250.737,A -85,B 0,C 180,E1 -8130.241,E2 -8130.241} C_VEL
LIN {X 0,Y 460.526,Z 250.741,A -85,B 0,C 180,E1 -8133.326,E2 -8133.326} C_VEL
LIN {X 0,Y 460.477,Z 250.745,A -85,B 0,C 180,E1 -8136.53,E2 -8136.53} C_VEL
LIN {X 0,Y 460.54,Z 250.74,A -85,B 0,C 180,E1 -8138.898,E2 -8138.898} C_VEL
LIN {X 0,Y 460.521,Z 250.744,A -85,B 0,C 180,E1 -8142.182,E2 -8142.182} C_VEL
LIN {X 0,Y 460.52,Z 250.745,A -85,B 0,C 180,E1 -8145.413,E2 -8145.413} C_VEL
LIN {X 0,Y 460.535,Z 250.74,A -85,B 0,C 180,E1 -8148.398,E2 -8148.398} C_VEL
LIN {X 0,Y 460.526,Z 250.725,A -85,B 0,C 180,E1 -8151.268,E2 -8151.268} C_VEL
LIN {X 0,Y 460.509,Z 250.746,A -85,B 0,C 180,E1 -8154.555,E2 -8154.555} C_VEL
LIN {X 0,Y 460.531,Z 250.746,A -85,B 0,C 180,E1 -8157.716,E2 -8157.716} C_VEL
LIN {X 0,Y 460.56,Z 250.944,A -85,B 0,C 180,E1 -8159.511,E2 -8159.511} C_VEL
LIN {X 0,Y 463.55,Z 263.653,A -85,B 0,C 180,E1 -8161.966,E2 -8161.966} C_VEL
LIN {X 0,Y 464.411,Z 269.311,A -85,B 0,C 180,E1 -8163,E2 -8163} C_VEL
LIN {X 0,Y 463.37,Z 287.564,A -85,B 0,C 180,E1 -8166.064,E2 -8166.064} C_VEL
LIN {X 0,Y 462.344,Z 307.232,A -85,B 0,C 180,E1 -8169.304,E2 -8169.304} C_VEL
LIN {X 0,Y 462.107,Z 313.919,A -85,B 0,C 180,E1 -8170.359,E2 -8170.359} C_VEL
LIN {X 0,Y 465.387,Z 333.471,A -85,B 0,C 180,E1 -8170.821,E2 -8170.821} C_VEL
LIN {X 0,Y 465.298,Z 351.201,A -85,B 0,C 180,E1 -8171.084,E2 -8171.084} C_VEL
LIN {X 0,Y 464.583,Z 357.054,A -85,B 0,C 180,E1 -8171.141,E2 -8171.141} C_VEL
LIN {X 0,Y 458.983,Z 376.087,A -85,B 0,C 180,E1 -8171.189,E2 -8171.189} C_VEL
LIN {X 0,Y 458.343,Z 381.936,A -85,B 0,C 180,E1 -8171.251,E2 -8171.251} C_VEL
LIN {X 0,Y 457.99,Z 425.912,A -85,B 0,C 180,E1 -8171.925,E2 -8171.925} C_VEL
LIN {X 0,Y 457.622,Z 439.018,A -85,B 0,C 180,E1 -8172.3,E2 -8172.3} C_VEL
LIN {X 0,Y 457.18,Z 451.899,A -85,B 0,C 180,E1 -8172.858,E2 -8172.858} C_VEL
LIN {X 0,Y 456.592,Z 463.948,A -85,B 0,C 180,E1 -8173.571,E2 -8173.571} C_VEL
LIN {X 0,Y 455.836,Z 475.517,A -85,B 0,C 180,E1 -8174.462,E2 -8174.462} C_VEL
LIN {X 0,Y 455.171,Z 485.906,A -85,B 0,C 180,E1 -8175.469,E2 -8175.469} C_VEL
LIN {X 0,Y 454.472,Z 495.278,A -85,B 0,C 180,E1 -8176.588,E2 -8176.588} C_VEL
LIN {X 0,Y 453.924,Z 504.304,A -85,B 0,C 180,E1 -8177.935,E2 -8177.935} C_VEL
LIN {X 0,Y 453.388,Z 511.576,A -85,B 0,C 180,E1 -8179.28,E2 -8179.28} C_VEL
LIN {X 0,Y 453.073,Z 517.419,A -85,B 0,C 180,E1 -8180.626,E2 -8180.626} C_VEL
LIN {X 0,Y 452.825,Z 522.053,A -85,B 0,C 180,E1 -8181.971,E2 -8181.971} C_VEL
LIN {X 0,Y 452.653,Z 526.188,A -85,B 0,C 180,E1 -8183.559,E2 -8183.559} C_VEL
LIN {X 0,Y 452.558,Z 528.221,A -85,B 0,C 180,E1 -8184.654,E2 -8184.654} C_VEL
LIN {X 0,Y 452.51,Z 530.312,A -85,B 0,C 180,E1 -8186.438,E2 -8186.438} C_VEL
LIN {X 0,Y 452.51,Z 530.786,A -85,B 0,C 180,E1 -8187.329,E2 -8187.329} C_VEL
LIN {X 0,Y 452.432,Z 530.589,A -85,B 0,C 180,E1 -8189.11,E2 -8189.11} C_VEL
LIN {X 0,Y 452.468,Z 528.941,A -85,B 0,C 180,E1 -8190.89,E2 -8190.89} C_VEL
LIN {X 0,Y 452.538,Z 527.521,A -85,B 0,C 180,E1 -8191.78,E2 -8191.78} C_VEL
LIN {X 0,Y 452.802,Z 523.449,A -85,B 0,C 180,E1 -8193.559,E2 -8193.559} C_VEL
LIN {X 0,Y 453.011,Z 519.229,A -85,B 0,C 180,E1 -8194.895,E2 -8194.895} C_VEL
LIN {X 0,Y 453.266,Z 512.893,A -85,B 0,C 180,E1 -8196.454,E2 -8196.454} C_VEL
LIN {X 0,Y 453.753,Z 506.257,A -85,B 0,C 180,E1 -8197.738,E2 -8197.738} C_VEL
LIN {X 0,Y 454.17,Z 498.947,A -85,B 0,C 180,E1 -8198.902,E2 -8198.902} C_VEL
LIN {X 0,Y 454.741,Z 490.465,A -85,B 0,C 180,E1 -8200.013,E2 -8200.013} C_VEL
LIN {X 0,Y 455.394,Z 480.041,A -85,B 0,C 180,E1 -8201.122,E2 -8201.122} C_VEL
LIN {X 0,Y 456.013,Z 469.701,A -85,B 0,C 180,E1 -8202.008,E2 -8202.008} C_VEL
LIN {X 0,Y 456.658,Z 458.335,A -85,B 0,C 180,E1 -8202.781,E2 -8202.781} C_VEL
LIN {X 0,Y 457.098,Z 446.608,A -85,B 0,C 180,E1 -8203.39,E2 -8203.39} C_VEL
LIN {X 0,Y 457.572,Z 432.983,A -85,B 0,C 180,E1 -8203.886,E2 -8203.886} C_VEL
LIN {X 0,Y 457.81,Z 420.72,A -85,B 0,C 180,E1 -8204.162,E2 -8204.162} C_VEL
LIN {X 0,Y 458.329,Z 333.003,A -85,B 0,C 180,E1 -8205.466,E2 -8205.466} C_VEL
LIN {X 0,Y 455.089,Z 313.962,A -85,B 0,C 180,E1 -8205.909,E2 -8205.909} C_VEL
LIN {X 0,Y 455.207,Z 310.033,A -85,B 0,C 180,E1 -8206.499,E2 -8206.499} C_VEL
LIN {X 0,Y 456.273,Z 288.836,A -85,B 0,C 180,E1 -8210.016,E2 -8210.016} C_VEL
LIN {X 0,Y 457.408,Z 269.479,A -85,B 0,C 180,E1 -8213.282,E2 -8213.282} C_VEL
LIN {X 0,Y 454.342,Z 255.269,A -85,B 0,C 180,E1 -8215.965,E2 -8215.965} C_VEL
LIN {X 0,Y 453.553,Z 251.683,A -85,B 0,C 180,E1 -8216.703,E2 -8216.703} C_VEL
LIN {X 0,Y 453.474,Z 251.611,A -85,B 0,C 180,E1 -8219.784,E2 -8219.784} C_VEL
LIN {X 0,Y 453.492,Z 251.607,A -85,B 0,C 180,E1 -8223.188,E2 -8223.188} C_VEL
LIN {X 0,Y 453.454,Z 251.625,A -85,B 0,C 180,E1 -8226.298,E2 -8226.298} C_VEL
LIN {X 0,Y 453.505,Z 251.621,A -85,B 0,C 180,E1 -8229.447,E2 -8229.447} C_VEL
LIN {X 0,Y 453.468,Z 251.625,A -85,B 0,C 180,E1 -8232.993,E2 -8232.993} C_VEL
LIN {X 0,Y 453.465,Z 251.62,A -85,B 0,C 180,E1 -8235.778,E2 -8235.778} C_VEL
LIN {X 0,Y 453.477,Z 251.619,A -85,B 0,C 180,E1 -8238.208,E2 -8238.208} C_VEL
LIN {X 0,Y 453.485,Z 251.61,A -85,B 0,C 180,E1 -8240.793,E2 -8240.793} C_VEL
LIN {X 0,Y 453.454,Z 251.621,A -85,B 0,C 180,E1 -8243.917,E2 -8243.917} C_VEL
LIN {X 0,Y 453.48,Z 251.612,A -85,B 0,C 180,E1 -8247.15,E2 -8247.15} C_VEL
LIN {X 0,Y 453.51,Z 251.616,A -85,B 0,C 180,E1 -8250.27,E2 -8250.27} C_VEL
LIN {X 0,Y 453.502,Z 251.62,A -85,B 0,C 180,E1 -8253.293,E2 -8253.293} C_VEL
LIN {X 0,Y 453.498,Z 251.612,A -85,B 0,C 180,E1 -8256.238,E2 -8256.238} C_VEL
LIN {X 0,Y 453.477,Z 251.62,A -85,B 0,C 180,E1 -8259.117,E2 -8259.117} C_VEL
LIN {X 0,Y 453.506,Z 251.615,A -85,B 0,C 180,E1 -8261.944,E2 -8261.944} C_VEL
LIN {X 0,Y 453.534,Z 251.613,A -85,B 0,C 180,E1 -8264.726,E2 -8264.726} C_VEL
LIN {X 0,Y 453.557,Z 251.61,A -85,B 0,C 180,E1 -8267.471,E2 -8267.471} C_VEL
LIN {X 0,Y 453.586,Z 251.607,A -85,B 0,C 180,E1 -8271.086,E2 -8271.086} C_VEL
LIN {X 0,Y 453.67,Z 251.595,A -85,B 0,C 180,E1 -8273.774,E2 -8273.774} C_VEL
LIN {X 0,Y 453.759,Z 251.584,A -85,B 0,C 180,E1 -8277.336,E2 -8277.336} C_VEL
LIN {X 0,Y 453.816,Z 251.577,A -85,B 0,C 180,E1 -8280,E2 -8280} C_VEL
LIN {X 0,Y 453.758,Z 251.589,A -85,B 0,C 180,E1 -8282.663,E2 -8282.663} C_VEL
LIN {X 0,Y 453.67,Z 251.594,A -85,B 0,C 180,E1 -8286.225,E2 -8286.225} C_VEL
LIN {X 0,Y 453.585,Z 251.606,A -85,B 0,C 180,E1 -8288.913,E2 -8288.913} C_VEL
LIN {X 0,Y 453.556,Z 251.614,A -85,B 0,C 180,E1 -8292.529,E2 -8292.529} C_VEL
LIN {X 0,Y 453.537,Z 251.612,A -85,B 0,C 180,E1 -8296.196,E2 -8296.196} C_VEL
LIN {X 0,Y 453.513,Z 251.614,A -85,B 0,C 180,E1 -8299.041,E2 -8299.041} C_VEL
LIN {X 0,Y 453.47,Z 251.622,A -85,B 0,C 180,E1 -8301.836,E2 -8301.836} C_VEL
LIN {X 0,Y 453.507,Z 251.613,A -85,B 0,C 180,E1 -8304.735,E2 -8304.735} C_VEL
LIN {X 0,Y 453.532,Z 251.615,A -85,B 0,C 180,E1 -8307.961,E2 -8307.961} C_VEL
LIN {X 0,Y 453.477,Z 251.608,A -85,B 0,C 180,E1 -8310.759,E2 -8310.759} C_VEL
LIN {X 0,Y 453.472,Z 251.628,A -85,B 0,C 180,E1 -8313.913,E2 -8313.913} C_VEL
LIN {X 0,Y 453.465,Z 251.61,A -85,B 0,C 180,E1 -8317.188,E2 -8317.188} C_VEL
LIN {X 0,Y 453.512,Z 251.619,A -85,B 0,C 180,E1 -8319.447,E2 -8319.447} C_VEL
LIN {X 0,Y 453.458,Z 251.618,A -85,B 0,C 180,E1 -8322.995,E2 -8322.995} C_VEL
LIN {X 0,Y 453.46,Z 251.618,A -85,B 0,C 180,E1 -8325.779,E2 -8325.779} C_VEL
LIN {X 0,Y 453.475,Z 251.594,A -85,B 0,C 180,E1 -8328.21,E2 -8328.21} C_VEL
LIN {X 0,Y 453.511,Z 251.616,A -85,B 0,C 180,E1 -8330.791,E2 -8330.791} C_VEL
LIN {X 0,Y 453.451,Z 251.607,A -85,B 0,C 180,E1 -8333.918,E2 -8333.918} C_VEL
LIN {X 0,Y 453.48,Z 251.62,A -85,B 0,C 180,E1 -8337.152,E2 -8337.152} C_VEL
LIN {X 0,Y 453.473,Z 251.624,A -85,B 0,C 180,E1 -8340.269,E2 -8340.269} C_VEL
LIN {X 0,Y 453.573,Z 251.756,A -85,B 0,C 180,E1 -8341.998,E2 -8341.998} C_VEL
LIN {X 0,Y 456.966,Z 266.102,A -85,B 0,C 180,E1 -8344.493,E2 -8344.493} C_VEL
LIN {X 0,Y 458.018,Z 271.286,A -85,B 0,C 180,E1 -8345.354,E2 -8345.354} C_VEL
LIN {X 0,Y 456.84,Z 289.64,A -85,B 0,C 180,E1 -8348.096,E2 -8348.096} C_VEL
LIN {X 0,Y 456.385,Z 297.094,A -85,B 0,C 180,E1 -8349.169,E2 -8349.169} C_VEL
LIN {X 0,Y 459.231,Z 315.674,A -85,B 0,C 180,E1 -8349.623,E2 -8349.623} C_VEL
LIN {X 0,Y 457.772,Z 432.563,A -85,B 0,C 180,E1 -8351.569,E2 -8351.569} C_VEL
LIN {X 0,Y 457.362,Z 446.883,A -85,B 0,C 180,E1 -8351.986,E2 -8351.986} C_VEL
LIN {X 0,Y 456.819,Z 460.431,A -85,B 0,C 180,E1 -8352.557,E2 -8352.557} C_VEL
LIN {X 0,Y 456.234,Z 474.105,A -85,B 0,C 180,E1 -8353.328,E2 -8353.328} C_VEL
LIN {X 0,Y 455.537,Z 486.597,A -85,B 0,C 180,E1 -8354.222,E2 -8354.222} C_VEL
LIN {X 0,Y 454.867,Z 498.02,A -85,B 0,C 180,E1 -8355.231,E2 -8355.231} C_VEL
LIN {X 0,Y 454.309,Z 508.518,A -85,B 0,C 180,E1 -8356.355,E2 -8356.355} C_VEL
LIN {X 0,Y 453.825,Z 518.921,A -85,B 0,C 180,E1 -8357.706,E2 -8357.706} C_VEL
LIN {X 0,Y 453.334,Z 527.505,A -85,B 0,C 180,E1 -8359.053,E2 -8359.053} C_VEL
LIN {X 0,Y 452.95,Z 535.685,A -85,B 0,C 180,E1 -8360.624,E2 -8360.624} C_VEL
LIN {X 0,Y 452.726,Z 541.425,A -85,B 0,C 180,E1 -8361.969,E2 -8361.969} C_VEL
LIN {X 0,Y 452.561,Z 547.13,A -85,B 0,C 180,E1 -8363.659,E2 -8363.659} C_VEL
LIN {X 0,Y 452.541,Z 549.791,A -85,B 0,C 180,E1 -8364.654,E2 -8364.654} C_VEL
LIN {X 0,Y 452.471,Z 553.385,A -85,B 0,C 180,E1 -8366.438,E2 -8366.438} C_VEL
LIN {X 0,Y 452.504,Z 554.634,A -85,B 0,C 180,E1 -8367.329,E2 -8367.329} C_VEL
LIN {X 0,Y 452.426,Z 556.066,A -85,B 0,C 180,E1 -8369.11,E2 -8369.11} C_VEL
LIN {X 0,Y 452.426,Z 556.09,A -85,B 0,C 180,E1 -8370.89,E2 -8370.89} C_VEL
LIN {X 0,Y 452.504,Z 554.701,A -85,B 0,C 180,E1 -8372.671,E2 -8372.671} C_VEL
LIN {X 0,Y 452.471,Z 551.884,A -85,B 0,C 180,E1 -8374.454,E2 -8374.454} C_VEL
LIN {X 0,Y 452.53,Z 548.826,A -85,B 0,C 180,E1 -8375.794,E2 -8375.794} C_VEL
LIN {X 0,Y 452.654,Z 544.818,A -85,B 0,C 180,E1 -8377.135,E2 -8377.135} C_VEL
LIN {X 0,Y 452.815,Z 539.868,A -85,B 0,C 180,E1 -8378.479,E2 -8378.479} C_VEL
LIN {X 0,Y 453.076,Z 532.713,A -85,B 0,C 180,E1 -8380.05,E2 -8380.05} C_VEL
LIN {X 0,Y 453.564,Z 523.84,A -85,B 0,C 180,E1 -8381.621,E2 -8381.621} C_VEL
LIN {X 0,Y 454.091,Z 514.42,A -85,B 0,C 180,E1 -8382.985,E2 -8382.985} C_VEL
LIN {X 0,Y 454.635,Z 504.262,A -85,B 0,C 180,E1 -8384.206,E2 -8384.206} C_VEL
LIN {X 0,Y 455.305,Z 492.932,A -85,B 0,C 180,E1 -8385.327,E2 -8385.327} C_VEL
LIN {X 0,Y 456.045,Z 480.381,A -85,B 0,C 180,E1 -8386.334,E2 -8386.334} C_VEL
LIN {X 0,Y 456.66,Z 468.406,A -85,B 0,C 180,E1 -8387.109,E2 -8387.109} C_VEL
LIN {X 0,Y 457.248,Z 454.078,A -85,B 0,C 180,E1 -8387.825,E2 -8387.825} C_VEL
LIN {X 0,Y 457.804,Z 439.587,A -85,B 0,C 180,E1 -8388.343,E2 -8388.343} C_VEL
LIN {X 0,Y 458.163,Z 424.812,A -85,B 0,C 180,E1 -8388.675,E2 -8388.675} C_VEL
LIN {X 0,Y 459.392,Z 314.223,A -85,B 0,C 180,E1 -8390.513,E2 -8390.513} C_VEL
LIN {X 0,Y 456.594,Z 297.264,A -85,B 0,C 180,E1 -8390.945,E2 -8390.945} C_VEL
LIN {X 0,Y 457.294,Z 285.933,A -85,B 0,C 180,E1 -8392.595,E2 -8392.595} C_VEL
LIN {X 0,Y 458.207,Z 272.164,A -85,B 0,C 180,E1 -8394.672,E2 -8394.672} C_VEL
LIN {X 0,Y 456.656,Z 264.207,A -85,B 0,C 180,E1 -8396.015,E2 -8396.015} C_VEL
LIN {X 0,Y 453.534,Z 251.718,A -85,B 0,C 180,E1 -8398.266,E2 -8398.266} C_VEL
LIN {X 0,Y 453.462,Z 251.608,A -85,B 0,C 180,E1 -8401.799,E2 -8401.799} C_VEL
LIN {X 0,Y 453.478,Z 251.616,A -85,B 0,C 180,E1 -8404.989,E2 -8404.989} C_VEL
LIN {X 0,Y 453.461,Z 251.62,A -85,B 0,C 180,E1 -8408.311,E2 -8408.311} C_VEL
LIN {X 0,Y 453.49,Z 251.618,A -85,B 0,C 180,E1 -8411.789,E2 -8411.789} C_VEL
LIN {X 0,Y 453.49,Z 251.615,A -85,B 0,C 180,E1 -8414.53,E2 -8414.53} C_VEL
LIN {X 0,Y 453.475,Z 251.616,A -85,B 0,C 180,E1 -8418.209,E2 -8418.209} C_VEL
LIN {X 0,Y 453.511,Z 251.618,A -85,B 0,C 180,E1 -8420.79,E2 -8420.79} C_VEL
LIN {X 0,Y 453.452,Z 251.615,A -85,B 0,C 180,E1 -8423.917,E2 -8423.917} C_VEL
LIN {X 0,Y 453.478,Z 251.62,A -85,B 0,C 180,E1 -8427.151,E2 -8427.151} C_VEL
LIN {X 0,Y 453.509,Z 251.604,A -85,B 0,C 180,E1 -8430.271,E2 -8430.271} C_VEL
LIN {X 0,Y 453.503,Z 251.617,A -85,B 0,C 180,E1 -8433.294,E2 -8433.294} C_VEL
LIN {X 0,Y 453.498,Z 251.621,A -85,B 0,C 180,E1 -8436.239,E2 -8436.239} C_VEL
LIN {X 0,Y 453.476,Z 251.618,A -85,B 0,C 180,E1 -8439.118,E2 -8439.118} C_VEL
LIN {X 0,Y 453.506,Z 251.62,A -85,B 0,C 180,E1 -8441.945,E2 -8441.945} C_VEL
LIN {X 0,Y 453.533,Z 251.611,A -85,B 0,C 180,E1 -8444.726,E2 -8444.726} C_VEL
LIN {X 0,Y 453.553,Z 251.607,A -85,B 0,C 180,E1 -8448.379,E2 -8448.379} C_VEL
LIN {X 0,Y 453.645,Z 251.596,A -85,B 0,C 180,E1 -8451.985,E2 -8451.985} C_VEL
LIN {X 0,Y 453.665,Z 251.596,A -85,B 0,C 180,E1 -8454.667,E2 -8454.667} C_VEL
LIN {X 0,Y 453.759,Z 251.585,A -85,B 0,C 180,E1 -8457.337,E2 -8457.337} C_VEL
LIN {X 0,Y 453.817,Z 251.579,A -85,B 0,C 180,E1 -8460,E2 -8460} C_VEL
LIN {X 0,Y 453.759,Z 251.579,A -85,B 0,C 180,E1 -8462.664,E2 -8462.664} C_VEL
LIN {X 0,Y 453.671,Z 251.592,A -85,B 0,C 180,E1 -8466.226,E2 -8466.226} C_VEL
LIN {X 0,Y 453.586,Z 251.607,A -85,B 0,C 180,E1 -8468.914,E2 -8468.914} C_VEL
LIN {X 0,Y 453.558,Z 251.607,A -85,B 0,C 180,E1 -8472.529,E2 -8472.529} C_VEL
LIN {X 0,Y 453.539,Z 251.608,A -85,B 0,C 180,E1 -8476.197,E2 -8476.197} C_VEL
LIN {X 0,Y 453.515,Z 251.62,A -85,B 0,C 180,E1 -8479.041,E2 -8479.041} C_VEL
LIN {X 0,Y 453.472,Z 251.622,A -85,B 0,C 180,E1 -8481.837,E2 -8481.837} C_VEL
LIN {X 0,Y 453.51,Z 251.616,A -85,B 0,C 180,E1 -8484.735,E2 -8484.735} C_VEL
LIN {X 0,Y 453.528,Z 251.605,A -85,B 0,C 180,E1 -8487.96,E2 -8487.96} C_VEL
LIN {X 0,Y 453.464,Z 251.624,A -85,B 0,C 180,E1 -8491.526,E2 -8491.526} C_VEL
LIN {X 0,Y 453.487,Z 251.612,A -85,B 0,C 180,E1 -8494.778,E2 -8494.778} C_VEL
LIN {X 0,Y 453.47,Z 251.622,A -85,B 0,C 180,E1 -8498.312,E2 -8498.312} C_VEL
LIN {X 0,Y 453.492,Z 251.612,A -85,B 0,C 180,E1 -8500.61,E2 -8500.61} C_VEL
LIN {X 0,Y 453.454,Z 251.62,A -85,B 0,C 180,E1 -8503.245,E2 -8503.245} C_VEL
LIN {X 0,Y 453.473,Z 251.622,A -85,B 0,C 180,E1 -8505.781,E2 -8505.781} C_VEL
LIN {X 0,Y 453.482,Z 251.617,A -85,B 0,C 180,E1 -8508.21,E2 -8508.21} C_VEL
LIN {X 0,Y 453.516,Z 251.603,A -85,B 0,C 180,E1 -8510.791,E2 -8510.791} C_VEL
LIN {X 0,Y 453.455,Z 251.626,A -85,B 0,C 180,E1 -8513.918,E2 -8513.918} C_VEL
LIN {X 0,Y 453.48,Z 251.618,A -85,B 0,C 180,E1 -8517.152,E2 -8517.152} C_VEL
LIN {X 0,Y 453.531,Z 251.785,A -85,B 0,C 180,E1 -8519.169,E2 -8519.169} C_VEL
LIN {X 0,Y 456.279,Z 263.485,A -85,B 0,C 180,E1 -8521.479,E2 -8521.479} C_VEL
LIN {X 0,Y 457.583,Z 270.807,A -85,B 0,C 180,E1 -8522.854,E2 -8522.854} C_VEL
LIN {X 0,Y 456.479,Z 288.829,A -85,B 0,C 180,E1 -8525.921,E2 -8525.921} C_VEL
LIN {X 0,Y 455.408,Z 308.51,A -85,B 0,C 180,E1 -8529.21,E2 -8529.21} C_VEL
LIN {X 0,Y 455.205,Z 313.828,A -85,B 0,C 180,E1 -8530.049,E2 -8530.049} C_VEL
LIN {X 0,Y 458.637,Z 333.322,A -85,B 0,C 180,E1 -8530.524,E2 -8530.524} C_VEL
LIN {X 0,Y 458.343,Z 381.936,A -85,B 0,C 180,E1 -8531.251,E2 -8531.251} C_VEL
LIN {X 0,Y 457.684,Z 387.79,A -85,B 0,C 180,E1 -8531.311,E2 -8531.311} C_VEL
LIN {X 0,Y 452.018,Z 406.814,A -85,B 0,C 180,E1 -8531.358,E2 -8531.358} C_VEL
LIN {X 0,Y 451.369,Z 412.667,A -85,B 0,C 180,E1 -8531.42,E2 -8531.42} C_VEL
LIN {X 0,Y 451.186,Z 429.585,A -85,B 0,C 180,E1 -8531.731,E2 -8531.731} C_VEL
LIN {X 0,Y 450.819,Z 441.157,A -85,B 0,C 180,E1 -8532.1,E2 -8532.1} C_VEL
LIN {X 0,Y 450.337,Z 453.592,A -85,B 0,C 180,E1 -8532.674,E2 -8532.674} C_VEL
LIN {X 0,Y 449.675,Z 465.644,A -85,B 0,C 180,E1 -8533.428,E2 -8533.428} C_VEL
LIN {X 0,Y 448.898,Z 476.919,A -85,B 0,C 180,E1 -8534.332,E2 -8534.332} C_VEL
LIN {X 0,Y 448.199,Z 487.084,A -85,B 0,C 180,E1 -8535.354,E2 -8535.354} C_VEL
LIN {X 0,Y 447.429,Z 496.951,A -85,B 0,C 180,E1 -8536.592,E2 -8536.592} C_VEL
LIN {X 0,Y 446.95,Z 504.439,A -85,B 0,C 180,E1 -8537.744,E2 -8537.744} C_VEL
LIN {X 0,Y 446.382,Z 511.716,A -85,B 0,C 180,E1 -8539.11,E2 -8539.11} C_VEL
LIN {X 0,Y 446.032,Z 517.566,A -85,B 0,C 180,E1 -8540.477,E2 -8540.477} C_VEL
LIN {X 0,Y 445.783,Z 522.207,A -85,B 0,C 180,E1 -8541.843,E2 -8541.843} C_VEL
LIN {X 0,Y 445.572,Z 526.594,A -85,B 0,C 180,E1 -8543.569,E2 -8543.569} C_VEL
LIN {X 0,Y 445.476,Z 528.393,A -85,B 0,C 180,E1 -8544.568,E2 -8544.568} C_VEL
LIN {X 0,Y 445.41,Z 530.495,A -85,B 0,C 180,E1 -8546.381,E2 -8546.381} C_VEL
LIN {X 0,Y 445.437,Z 530.979,A -85,B 0,C 180,E1 -8547.287,E2 -8547.287} C_VEL
LIN {X 0,Y 445.342,Z 530.799,A -85,B 0,C 180,E1 -8549.096,E2 -8549.096} C_VEL
LIN {X 0,Y 445.377,Z 529.169,A -85,B 0,C 180,E1 -8550.904,E2 -8550.904} C_VEL
LIN {X 0,Y 445.453,Z 527.768,A -85,B 0,C 180,E1 -8551.808,E2 -8551.808} C_VEL
LIN {X 0,Y 445.739,Z 523.718,A -85,B 0,C 180,E1 -8553.616,E2 -8553.616} C_VEL
LIN {X 0,Y 445.953,Z 519.524,A -85,B 0,C 180,E1 -8554.972,E2 -8554.972} C_VEL
LIN {X 0,Y 446.243,Z 513.223,A -85,B 0,C 180,E1 -8556.556,E2 -8556.556} C_VEL
LIN {X 0,Y 446.705,Z 506.91,A -85,B 0,C 180,E1 -8557.81,E2 -8557.81} C_VEL
LIN {X 0,Y 447.17,Z 499.367,A -85,B 0,C 180,E1 -8559.042,E2 -8559.042} C_VEL
LIN {X 0,Y 447.785,Z 490.941,A -85,B 0,C 180,E1 -8560.17,E2 -8560.17} C_VEL
LIN {X 0,Y 448.467,Z 480.584,A -85,B 0,C 180,E1 -8561.296,E2 -8561.296} C_VEL
LIN {X 0,Y 449.121,Z 470.332,A -85,B 0,C 180,E1 -8562.195,E2 -8562.195} C_VEL
LIN {X 0,Y 449.77,Z 459.098,A -85,B 0,C 180,E1 -8562.98,E2 -8562.98} C_VEL
LIN {X 0,Y 450.257,Z 447.648,A -85,B 0,C 180,E1 -8563.598,E2 -8563.598} C_VEL
LIN {X 0,Y 450.756,Z 434.453,A -85,B 0,C 180,E1 -8564.1,E2 -8564.1} C_VEL
LIN {X 0,Y 451.019,Z 421.577,A -85,B 0,C 180,E1 -8564.408,E2 -8564.408} C_VEL
LIN {X 0,Y 451.536,Z 333.568,A -85,B 0,C 180,E1 -8565.74,E2 -8565.74} C_VEL
LIN {X 0,Y 448.148,Z 313.614,A -85,B 0,C 180,E1 -8566.221,E2 -8566.221} C_VEL
LIN {X 0,Y 449.118,Z 294.333,A -85,B 0,C 180,E1 -8569.422,E2 -8569.422} C_VEL
LIN {X 0,Y 450.374,Z 273.528,A -85,B 0,C 180,E1 -8572.972,E2 -8572.972} C_VEL
LIN {X 0,Y 450.551,Z 271.101,A -85,B 0,C 180,E1 -8573.389,E2 -8573.389} C_VEL
LIN {X 0,Y 447.18,Z 255.523,A -85,B 0,C 180,E1 -8576.384,E2 -8576.384} C_VEL
LIN {X 0,Y 446.509,Z 252.604,A -85,B 0,C 180,E1 -8576.986,E2 -8576.986} C_VEL
LIN {X 0,Y 446.429,Z 252.49,A -85,B 0,C 180,E1 -8580.249,E2 -8580.249} C_VEL
LIN {X 0,Y 446.446,Z 252.482,A -85,B 0,C 180,E1 -8583.453,E2 -8583.453} C_VEL
LIN {X 0,Y 446.402,Z 252.505,A -85,B 0,C 180,E1 -8586.744,E2 -8586.744} C_VEL
LIN {X 0,Y 446.468,Z 252.497,A -85,B 0,C 180,E1 -8589.526,E2 -8589.526} C_VEL
LIN {X 0,Y 446.432,Z 252.498,A -85,B 0,C 180,E1 -8592.603,E2 -8592.603} C_VEL
LIN {X 0,Y 446.453,Z 252.491,A -85,B 0,C 180,E1 -8595.102,E2 -8595.102} C_VEL
LIN {X 0,Y 446.426,Z 252.5,A -85,B 0,C 180,E1 -8598.608,E2 -8598.608} C_VEL
LIN {X 0,Y 446.437,Z 252.489,A -85,B 0,C 180,E1 -8600.972,E2 -8600.972} C_VEL
LIN {X 0,Y 446.418,Z 252.499,A -85,B 0,C 180,E1 -8604.373,E2 -8604.373} C_VEL
LIN {X 0,Y 446.419,Z 252.495,A -85,B 0,C 180,E1 -8607.638,E2 -8607.638} C_VEL
LIN {X 0,Y 446.465,Z 252.498,A -85,B 0,C 180,E1 -8610.791,E2 -8610.791} C_VEL
LIN {X 0,Y 446.473,Z 252.492,A -85,B 0,C 180,E1 -8613.848,E2 -8613.848} C_VEL
LIN {X 0,Y 446.424,Z 252.5,A -85,B 0,C 180,E1 -8616.823,E2 -8616.823} C_VEL
LIN {X 0,Y 446.438,Z 252.492,A -85,B 0,C 180,E1 -8619.736,E2 -8619.736} C_VEL
LIN {X 0,Y 446.458,Z 252.499,A -85,B 0,C 180,E1 -8622.597,E2 -8622.597} C_VEL
LIN {X 0,Y 446.466,Z 252.489,A -85,B 0,C 180,E1 -8625.412,E2 -8625.412} C_VEL
LIN {X 0,Y 446.511,Z 252.49,A -85,B 0,C 180,E1 -8628.193,E2 -8628.193} C_VEL
LIN {X 0,Y 446.594,Z 252.476,A -85,B 0,C 180,E1 -8631.857,E2 -8631.857} C_VEL
LIN {X 0,Y 446.639,Z 252.471,A -85,B 0,C 180,E1 -8634.582,E2 -8634.582} C_VEL
LIN {X 0,Y 446.703,Z 252.463,A -85,B 0,C 180,E1 -8637.294,E2 -8637.294} C_VEL
LIN {X 0,Y 446.786,Z 252.453,A -85,B 0,C 180,E1 -8640,E2 -8640} C_VEL
LIN {X 0,Y 446.702,Z 252.468,A -85,B 0,C 180,E1 -8642.705,E2 -8642.705} C_VEL
LIN {X 0,Y 446.639,Z 252.47,A -85,B 0,C 180,E1 -8646.324,E2 -8646.324} C_VEL
LIN {X 0,Y 446.531,Z 252.484,A -85,B 0,C 180,E1 -8649.055,E2 -8649.055} C_VEL
LIN {X 0,Y 446.514,Z 252.489,A -85,B 0,C 180,E1 -8652.73,E2 -8652.73} C_VEL
LIN {X 0,Y 446.489,Z 252.49,A -85,B 0,C 180,E1 -8656.228,E2 -8656.228} C_VEL
LIN {X 0,Y 446.462,Z 252.493,A -85,B 0,C 180,E1 -8659.303,E2 -8659.303} C_VEL
LIN {X 0,Y 446.413,Z 252.506,A -85,B 0,C 180,E1 -8662.2,E2 -8662.2} C_VEL
LIN {X 0,Y 446.451,Z 252.491,A -85,B 0,C 180,E1 -8665.153,E2 -8665.153} C_VEL
LIN {X 0,Y 446.478,Z 252.49,A -85,B 0,C 180,E1 -8668.179,E2 -8668.179} C_VEL
LIN {X 0,Y 446.414,Z 252.488,A -85,B 0,C 180,E1 -8671.3,E2 -8671.3} C_VEL
LIN {X 0,Y 446.425,Z 252.499,A -85,B 0,C 180,E1 -8674.523,E2 -8674.523} C_VEL
LIN {X 0,Y 446.425,Z 252.498,A -85,B 0,C 180,E1 -8678.082,E2 -8678.082} C_VEL
LIN {X 0,Y 446.422,Z 252.498,A -85,B 0,C 180,E1 -8680.918,E2 -8680.918} C_VEL
LIN {X 0,Y 446.413,Z 252.505,A -85,B 0,C 180,E1 -8683.844,E2 -8683.844} C_VEL
LIN {X 0,Y 446.394,Z 252.491,A -85,B 0,C 180,E1 -8686.404,E2 -8686.404} C_VEL
LIN {X 0,Y 446.423,Z 252.478,A -85,B 0,C 180,E1 -8689.083,E2 -8689.083} C_VEL
LIN {X 0,Y 446.412,Z 252.502,A -85,B 0,C 180,E1 -8691.921,E2 -8691.921} C_VEL
LIN {X 0,Y 446.426,Z 252.493,A -85,B 0,C 180,E1 -8695.478,E2 -8695.478} C_VEL
LIN {X 0,Y 446.414,Z 252.488,A -85,B 0,C 180,E1 -8698.7,E2 -8698.7} C_VEL
LIN {X 0,Y 446.525,Z 252.672,A -85,B 0,C 180,E1 -8701.681,E2 -8701.681} C_VEL
LIN {X 0,Y 450.029,Z 267.352,A -85,B 0,C 180,E1 -8704.281,E2 -8704.281} C_VEL
LIN {X 0,Y 451.119,Z 272.318,A -85,B 0,C 180,E1 -8705.126,E2 -8705.126} C_VEL
LIN {X 0,Y 450.335,Z 285.793,A -85,B 0,C 180,E1 -8707.181,E2 -8707.181} C_VEL
LIN {X 0,Y 449.52,Z 297.131,A -85,B 0,C 180,E1 -8708.865,E2 -8708.865} C_VEL
LIN {X 0,Y 452.507,Z 316.514,A -85,B 0,C 180,E1 -8709.355,E2 -8709.355} C_VEL
LIN {X 0,Y 450.97,Z 432.308,A -85,B 0,C 180,E1 -8711.31,E2 -8711.31} C_VEL
LIN {X 0,Y 450.539,Z 446.679,A -85,B 0,C 180,E1 -8711.733,E2 -8711.733} C_VEL
LIN {X 0,Y 449.932,Z 461.063,A -85,B 0,C 180,E1 -8712.352,E2 -8712.352} C_VEL
LIN {X 0,Y 449.362,Z 473.493,A -85,B 0,C 180,E1 -8713.065,E2 -8713.065} C_VEL
LIN {X 0,Y 448.653,Z 486.079,A -85,B 0,C 180,E1 -8713.973,E2 -8713.973} C_VEL
LIN {X 0,Y 447.949,Z 497.568,A -85,B 0,C 180,E1 -8714.997,E2 -8714.997} C_VEL
LIN {X 0,Y 447.321,Z 508.116,A -85,B 0,C 180,E1 -8716.138,E2 -8716.138} C_VEL
LIN {X 0,Y 446.833,Z 518.579,A -85,B 0,C 180,E1 -8717.51,E2 -8717.51} C_VEL
LIN {X 0,Y 446.302,Z 527.193,A -85,B 0,C 180,E1 -8718.878,E2 -8718.878} C_VEL
LIN {X 0,Y 445.896,Z 535.399,A -85,B 0,C 180,E1 -8720.474,E2 -8720.474} C_VEL
LIN {X 0,Y 445.648,Z 541.161,A -85,B 0,C 180,E1 -8721.841,E2 -8721.841} C_VEL
LIN {X 0,Y 445.54,Z 545.847,A -85,B 0,C 180,E1 -8723.206,E2 -8723.206} C_VEL
LIN {X 0,Y 445.434,Z 549.555,A -85,B 0,C 180,E1 -8724.568,E2 -8724.568} C_VEL
LIN {X 0,Y 445.369,Z 553.164,A -85,B 0,C 180,E1 -8726.381,E2 -8726.381} C_VEL
LIN {X 0,Y 445.429,Z 554.42,A -85,B 0,C 180,E1 -8727.287,E2 -8727.287} C_VEL
LIN {X 0,Y 445.336,Z 555.861,A -85,B 0,C 180,E1 -8729.096,E2 -8729.096} C_VEL
LIN {X 0,Y 445.336,Z 555.894,A -85,B 0,C 180,E1 -8730.904,E2 -8730.904} C_VEL
LIN {X 0,Y 445.429,Z 554.511,A -85,B 0,C 180,E1 -8732.713,E2 -8732.713} C_VEL
LIN {X 0,Y 445.392,Z 551.695,A -85,B 0,C 180,E1 -8734.525,E2 -8734.525} C_VEL
LIN {X 0,Y 445.488,Z 547.383,A -85,B 0,C 180,E1 -8736.34,E2 -8736.34} C_VEL
LIN {X 0,Y 445.614,Z 543.103,A -85,B 0,C 180,E1 -8737.704,E2 -8737.704} C_VEL
LIN {X 0,Y 445.871,Z 536.809,A -85,B 0,C 180,E1 -8739.298,E2 -8739.298} C_VEL
LIN {X 0,Y 446.284,Z 528.942,A -85,B 0,C 180,E1 -8740.893,E2 -8740.893} C_VEL
LIN {X 0,Y 446.706,Z 520.715,A -85,B 0,C 180,E1 -8742.263,E2 -8742.263} C_VEL
LIN {X 0,Y 447.287,Z 510.783,A -85,B 0,C 180,E1 -8743.632,E2 -8743.632} C_VEL
LIN {X 0,Y 447.945,Z 499.741,A -85,B 0,C 180,E1 -8744.887,E2 -8744.887} C_VEL
LIN {X 0,Y 448.754,Z 487.466,A -85,B 0,C 180,E1 -8746.023,E2 -8746.023} C_VEL
LIN {X 0,Y 449.48,Z 475.275,A -85,B 0,C 180,E1 -8746.931,E2 -8746.931} C_VEL
LIN {X 0,Y 450.153,Z 462.271,A -85,B 0,C 180,E1 -8747.697,E2 -8747.697} C_VEL
LIN {X 0,Y 450.709,Z 448.365,A -85,B 0,C 180,E1 -8748.318,E2 -8748.318} C_VEL
LIN {X 0,Y 451.235,Z 433.788,A -85,B 0,C 180,E1 -8748.767,E2 -8748.767} C_VEL
LIN {X 0,Y 451.711,Z 403.678,A -85,B 0,C 180,E1 -8749.306,E2 -8749.306} C_VEL
LIN {X 0,Y 452.655,Z 314.575,A -85,B 0,C 180,E1 -8750.813,E2 -8750.813} C_VEL
LIN {X 0,Y 449.752,Z 297.185,A -85,B 0,C 180,E1 -8751.28,E2 -8751.28} C_VEL
LIN {X 0,Y 451.115,Z 278.258,A -85,B 0,C 180,E1 -8754.139,E2 -8754.139} C_VEL
LIN {X 0,Y 451.4,Z 273.592,A -85,B 0,C 180,E1 -8754.858,E2 -8754.858} C_VEL
LIN {X 0,Y 448.956,Z 262.211,A -85,B 0,C 180,E1 -8756.839,E2 -8756.839} C_VEL
LIN {X 0,Y 446.495,Z 252.582,A -85,B 0,C 180,E1 -8758.637,E2 -8758.637} C_VEL
LIN {X 0,Y 446.42,Z 252.486,A -85,B 0,C 180,E1 -8762.361,E2 -8762.361} C_VEL
LIN {X 0,Y 446.416,Z 252.486,A -85,B 0,C 180,E1 -8765.626,E2 -8765.626} C_VEL
LIN {X 0,Y 446.441,Z 252.499,A -85,B 0,C 180,E1 -8769.027,E2 -8769.027} C_VEL
LIN {X 0,Y 446.448,Z 252.501,A -85,B 0,C 180,E1 -8772.279,E2 -8772.279} C_VEL
LIN {X 0,Y 446.451,Z 252.492,A -85,B 0,C 180,E1 -8775.103,E2 -8775.103} C_VEL
LIN {X 0,Y 446.424,Z 252.491,A -85,B 0,C 180,E1 -8778.609,E2 -8778.609} C_VEL
LIN {X 0,Y 446.456,Z 252.496,A -85,B 0,C 180,E1 -8780.974,E2 -8780.974} C_VEL
LIN {X 0,Y 446.416,Z 252.492,A -85,B 0,C 180,E1 -8784.374,E2 -8784.374} C_VEL
LIN {X 0,Y 446.418,Z 252.502,A -85,B 0,C 180,E1 -8787.638,E2 -8787.638} C_VEL
LIN {X 0,Y 446.464,Z 252.483,A -85,B 0,C 180,E1 -8790.792,E2 -8790.792} C_VEL
LIN {X 0,Y 446.472,Z 252.498,A -85,B 0,C 180,E1 -8793.848,E2 -8793.848} C_VEL
LIN {X 0,Y 446.423,Z 252.498,A -85,B 0,C 180,E1 -8796.823,E2 -8796.823} C_VEL
LIN {X 0,Y 446.438,Z 252.497,A -85,B 0,C 180,E1 -8799.737,E2 -8799.737} C_VEL
LIN {X 0,Y 446.457,Z 252.492,A -85,B 0,C 180,E1 -8802.597,E2 -8802.597} C_VEL
LIN {X 0,Y 446.464,Z 252.494,A -85,B 0,C 180,E1 -8805.412,E2 -8805.412} C_VEL
LIN {X 0,Y 446.511,Z 252.485,A -85,B 0,C 180,E1 -8808.193,E2 -8808.193} C_VEL
LIN {X 0,Y 446.594,Z 252.476,A -85,B 0,C 180,E1 -8811.858,E2 -8811.858} C_VEL
LIN {X 0,Y 446.639,Z 252.471,A -85,B 0,C 180,E1 -8814.583,E2 -8814.583} C_VEL
LIN {X 0,Y 446.703,Z 252.463,A -85,B 0,C 180,E1 -8817.295,E2 -8817.295} C_VEL
LIN {X 0,Y 446.787,Z 252.455,A -85,B 0,C 180,E1 -8820,E2 -8820} C_VEL
LIN {X 0,Y 446.703,Z 252.458,A -85,B 0,C 180,E1 -8822.706,E2 -8822.706} C_VEL
LIN {X 0,Y 446.64,Z 252.467,A -85,B 0,C 180,E1 -8826.324,E2 -8826.324} C_VEL
LIN {X 0,Y 446.532,Z 252.487,A -85,B 0,C 180,E1 -8829.056,E2 -8829.056} C_VEL
LIN {X 0,Y 446.516,Z 252.485,A -85,B 0,C 180,E1 -8832.73,E2 -8832.73} C_VEL
LIN {X 0,Y 446.491,Z 252.486,A -85,B 0,C 180,E1 -8836.228,E2 -8836.228} C_VEL
LIN {X 0,Y 446.464,Z 252.494,A -85,B 0,C 180,E1 -8839.304,E2 -8839.304} C_VEL
LIN {X 0,Y 446.413,Z 252.5,A -85,B 0,C 180,E1 -8842.2,E2 -8842.2} C_VEL
LIN {X 0,Y 446.454,Z 252.5,A -85,B 0,C 180,E1 -8845.153,E2 -8845.153} C_VEL
LIN {X 0,Y 446.481,Z 252.483,A -85,B 0,C 180,E1 -8848.179,E2 -8848.179} C_VEL
LIN {X 0,Y 446.417,Z 252.501,A -85,B 0,C 180,E1 -8851.776,E2 -8851.776} C_VEL
LIN {X 0,Y 446.428,Z 252.493,A -85,B 0,C 180,E1 -8854.524,E2 -8854.524} C_VEL
LIN {X 0,Y 446.428,Z 252.499,A -85,B 0,C 180,E1 -8858.082,E2 -8858.082} C_VEL
LIN {X 0,Y 446.425,Z 252.496,A -85,B 0,C 180,E1 -8860.918,E2 -8860.918} C_VEL
LIN {X 0,Y 446.401,Z 252.496,A -85,B 0,C 180,E1 -8863.847,E2 -8863.847} C_VEL
LIN {X 0,Y 446.421,Z 252.504,A -85,B 0,C 180,E1 -8866.401,E2 -8866.401} C_VEL
LIN {X 0,Y 446.452,Z 252.496,A -85,B 0,C 180,E1 -8869.804,E2 -8869.804} C_VEL
LIN {X 0,Y 446.409,Z 252.48,A -85,B 0,C 180,E1 -8872.122,E2 -8872.122} C_VEL
LIN {X 0,Y 446.424,Z 252.488,A -85,B 0,C 180,E1 -8875.477,E2 -8875.477} C_VEL
LIN {X 0,Y 446.485,Z 252.715,A -85,B 0,C 180,E1 -8878.838,E2 -8878.838} C_VEL
LIN {X 0,Y 449.731,Z 266.471,A -85,B 0,C 180,E1 -8881.591,E2 -8881.591} C_VEL
LIN {X 0,Y 450.75,Z 272.381,A -85,B 0,C 180,E1 -8882.716,E2 -8882.716} C_VEL
LIN {X 0,Y 449.608,Z 290.098,A -85,B 0,C 180,E1 -8885.775,E2 -8885.775} C_VEL
LIN {X 0,Y 448.446,Z 309.921,A -85,B 0,C 180,E1 -8889.137,E2 -8889.137} C_VEL
LIN {X 0,Y 448.329,Z 313.757,A -85,B 0,C 180,E1 -8889.73,E2 -8889.73} C_VEL
LIN {X 0,Y 452.04,Z 335.22,A -85,B 0,C 180,E1 -8890.255,E2 -8890.255} C_VEL
LIN {X 0,Y 451.369,Z 412.667,A -85,B 0,C 180,E1 -8891.42,E2 -8891.42} C_VEL
LIN {X 0,Y 450.698,Z 418.523,A -85,B 0,C 180,E1 -8891.48,E2 -8891.48} C_VEL
LIN {X 0,Y 447.808,Z 428.015,A -85,B 0,C 180,E1 -8891.547,E2 -8891.547} C_VEL
LIN {X 0,Y 444.851,Z 437.379,A -85,B 0,C 180,E1 -8891.7,E2 -8891.7} C_VEL
LIN {X 0,Y 444.037,Z 443.023,A -85,B 0,C 180,E1 -8891.89,E2 -8891.89} C_VEL
LIN {X 0,Y 443.491,Z 455.027,A -85,B 0,C 180,E1 -8892.477,E2 -8892.477} C_VEL
LIN {X 0,Y 442.779,Z 467.336,A -85,B 0,C 180,E1 -8893.281,E2 -8893.281} C_VEL
LIN {X 0,Y 441.967,Z 478.309,A -85,B 0,C 180,E1 -8894.198,E2 -8894.198} C_VEL
LIN {X 0,Y 441.225,Z 488.193,A -85,B 0,C 180,E1 -8895.235,E2 -8895.235} C_VEL
LIN {X 0,Y 440.469,Z 497.32,A -85,B 0,C 180,E1 -8896.412,E2 -8896.412} C_VEL
LIN {X 0,Y 439.892,Z 505.901,A -85,B 0,C 180,E1 -8897.779,E2 -8897.779} C_VEL
LIN {X 0,Y 439.313,Z 512.947,A -85,B 0,C 180,E1 -8899.166,E2 -8899.166} C_VEL
LIN {X 0,Y 438.89,Z 519.393,A -85,B 0,C 180,E1 -8900.786,E2 -8900.786} C_VEL
LIN {X 0,Y 438.667,Z 523.676,A -85,B 0,C 180,E1 -8902.173,E2 -8902.173} C_VEL
LIN {X 0,Y 438.467,Z 527.031,A -85,B 0,C 180,E1 -8903.607,E2 -8903.607} C_VEL
LIN {X 0,Y 438.322,Z 529.808,A -85,B 0,C 180,E1 -8905.402,E2 -8905.402} C_VEL
LIN {X 0,Y 438.364,Z 531.172,A -85,B 0,C 180,E1 -8907.243,E2 -8907.243} C_VEL
LIN {X 0,Y 438.256,Z 531.008,A -85,B 0,C 180,E1 -8909.081,E2 -8909.081} C_VEL
LIN {X 0,Y 438.29,Z 529.395,A -85,B 0,C 180,E1 -8910.919,E2 -8910.919} C_VEL
LIN {X 0,Y 438.372,Z 528.013,A -85,B 0,C 180,E1 -8911.837,E2 -8911.837} C_VEL
LIN {X 0,Y 438.679,Z 523.985,A -85,B 0,C 180,E1 -8913.674,E2 -8913.674} C_VEL
LIN {X 0,Y 438.877,Z 519.817,A -85,B 0,C 180,E1 -8915.053,E2 -8915.053} C_VEL
LIN {X 0,Y 439.134,Z 514.524,A -85,B 0,C 180,E1 -8916.432,E2 -8916.432} C_VEL
LIN {X 0,Y 439.649,Z 507.929,A -85,B 0,C 180,E1 -8917.809,E2 -8917.809} C_VEL
LIN {X 0,Y 440.187,Z 499.771,A -85,B 0,C 180,E1 -8919.187,E2 -8919.187} C_VEL
LIN {X 0,Y 440.835,Z 491.406,A -85,B 0,C 180,E1 -8920.332,E2 -8920.332} C_VEL
LIN {X 0,Y 441.539,Z 481.117,A -85,B 0,C 180,E1 -8921.476,E2 -8921.476} C_VEL
LIN {X 0,Y 442.231,Z 470.95,A -85,B 0,C 180,E1 -8922.388,E2 -8922.388} C_VEL
LIN {X 0,Y 442.907,Z 459.836,A -85,B 0,C 180,E1 -8923.185,E2 -8923.185} C_VEL
LIN {X 0,Y 443.454,Z 447.41,A -85,B 0,C 180,E1 -8923.869,E2 -8923.869} C_VEL
LIN {X 0,Y 443.988,Z 434.041,A -85,B 0,C 180,E1 -8924.378,E2 -8924.378} C_VEL
LIN {X 0,Y 444.244,Z 421.11,A -85,B 0,C 180,E1 -8924.686,E2 -8924.686} C_VEL
LIN {X 0,Y 444.829,Z 334.459,A -85,B 0,C 180,E1 -8926.014,E2 -8926.014} C_VEL
LIN {X 0,Y 441.257,Z 313.628,A -85,B 0,C 180,E1 -8926.518,E2 -8926.518} C_VEL
LIN {X 0,Y 441.544,Z 306.927,A -85,B 0,C 180,E1 -8927.603,E2 -8927.603} C_VEL
LIN {X 0,Y 442.659,Z 287.534,A -85,B 0,C 180,E1 -8930.93,E2 -8930.93} C_VEL
LIN {X 0,Y 443.587,Z 272.313,A -85,B 0,C 180,E1 -8933.581,E2 -8933.581} C_VEL
LIN {X 0,Y 440.241,Z 256.765,A -85,B 0,C 180,E1 -8936.621,E2 -8936.621} C_VEL
LIN {X 0,Y 439.451,Z 253.437,A -85,B 0,C 180,E1 -8937.34,E2 -8937.34} C_VEL
LIN {X 0,Y 439.363,Z 253.376,A -85,B 0,C 180,E1 -8940.788,E2 -8940.788} C_VEL
LIN {X 0,Y 439.388,Z 253.361,A -85,B 0,C 180,E1 -8944.043,E2 -8944.043} C_VEL
LIN {X 0,Y 439.349,Z 253.385,A -85,B 0,C 180,E1 -8946.886,E2 -8946.886} C_VEL
LIN {X 0,Y 439.406,Z 253.373,A -85,B 0,C 180,E1 -8949.849,E2 -8949.849} C_VEL
LIN {X 0,Y 439.385,Z 253.376,A -85,B 0,C 180,E1 -8952.627,E2 -8952.627} C_VEL
LIN {X 0,Y 439.401,Z 253.369,A -85,B 0,C 180,E1 -8955.27,E2 -8955.27} C_VEL
LIN {X 0,Y 439.386,Z 253.378,A -85,B 0,C 180,E1 -8958.742,E2 -8958.742} C_VEL
LIN {X 0,Y 439.377,Z 253.377,A -85,B 0,C 180,E1 -8961.606,E2 -8961.606} C_VEL
LIN {X 0,Y 439.398,Z 253.37,A -85,B 0,C 180,E1 -8964.843,E2 -8964.843} C_VEL
LIN {X 0,Y 439.371,Z 253.372,A -85,B 0,C 180,E1 -8968.139,E2 -8968.139} C_VEL
LIN {X 0,Y 439.421,Z 253.369,A -85,B 0,C 180,E1 -8971.326,E2 -8971.326} C_VEL
LIN {X 0,Y 439.401,Z 253.376,A -85,B 0,C 180,E1 -8974.414,E2 -8974.414} C_VEL
LIN {X 0,Y 439.36,Z 253.38,A -85,B 0,C 180,E1 -8977.424,E2 -8977.424} C_VEL
LIN {X 0,Y 439.436,Z 253.368,A -85,B 0,C 180,E1 -8980.662,E2 -8980.662} C_VEL
LIN {X 0,Y 439.457,Z 253.367,A -85,B 0,C 180,E1 -8984.224,E2 -8984.224} C_VEL
LIN {X 0,Y 439.477,Z 253.364,A -85,B 0,C 180,E1 -8988.001,E2 -8988.001} C_VEL
LIN {X 0,Y 439.541,Z 253.354,A -85,B 0,C 180,E1 -8991.726,E2 -8991.726} C_VEL
LIN {X 0,Y 439.614,Z 253.347,A -85,B 0,C 180,E1 -8994.495,E2 -8994.495} C_VEL
LIN {X 0,Y 439.629,Z 253.348,A -85,B 0,C 180,E1 -8998.167,E2 -8998.167} C_VEL
LIN {X 0,Y 439.756,Z 253.329,A -85,B 0,C 180,E1 -9000,E2 -9000} C_VEL
LIN {X 0,Y 439.649,Z 253.346,A -85,B 0,C 180,E1 -9002.748,E2 -9002.748} C_VEL
LIN {X 0,Y 439.611,Z 253.346,A -85,B 0,C 180,E1 -9006.425,E2 -9006.425} C_VEL
LIN {X 0,Y 439.493,Z 253.361,A -85,B 0,C 180,E1 -9009.202,E2 -9009.202} C_VEL
LIN {X 0,Y 439.459,Z 253.367,A -85,B 0,C 180,E1 -9012.938,E2 -9012.938} C_VEL
LIN {X 0,Y 439.44,Z 253.369,A -85,B 0,C 180,E1 -9016.349,E2 -9016.349} C_VEL
LIN {X 0,Y 439.395,Z 253.375,A -85,B 0,C 180,E1 -9019.626,E2 -9019.626} C_VEL
LIN {X 0,Y 439.359,Z 253.381,A -85,B 0,C 180,E1 -9022.576,E2 -9022.576} C_VEL
LIN {X 0,Y 439.398,Z 253.372,A -85,B 0,C 180,E1 -9025.585,E2 -9025.585} C_VEL
LIN {X 0,Y 439.419,Z 253.365,A -85,B 0,C 180,E1 -9028.673,E2 -9028.673} C_VEL
LIN {X 0,Y 439.369,Z 253.371,A -85,B 0,C 180,E1 -9031.861,E2 -9031.861} C_VEL
LIN {X 0,Y 439.395,Z 253.374,A -85,B 0,C 180,E1 -9035.156,E2 -9035.156} C_VEL
LIN {X 0,Y 439.385,Z 253.376,A -85,B 0,C 180,E1 -9038.595,E2 -9038.595} C_VEL
LIN {X 0,Y 439.383,Z 253.376,A -85,B 0,C 180,E1 -9041.257,E2 -9041.257} C_VEL
LIN {X 0,Y 439.399,Z 253.374,A -85,B 0,C 180,E1 -9044.729,E2 -9044.729} C_VEL
LIN {X 0,Y 439.392,Z 253.347,A -85,B 0,C 180,E1 -9047.796,E2 -9047.796} C_VEL
LIN {X 0,Y 439.433,Z 253.367,A -85,B 0,C 180,E1 -9050.229,E2 -9050.229} C_VEL
LIN {X 0,Y 439.37,Z 253.361,A -85,B 0,C 180,E1 -9053.713,E2 -9053.713} C_VEL
LIN {X 0,Y 439.37,Z 253.378,A -85,B 0,C 180,E1 -9057.055,E2 -9057.055} C_VEL
LIN {X 0,Y 439.417,Z 253.367,A -85,B 0,C 180,E1 -9060.804,E2 -9060.804} C_VEL
LIN {X 0,Y 439.491,Z 253.6,A -85,B 0,C 180,E1 -9061.357,E2 -9061.357} C_VEL
LIN {X 0,Y 442.847,Z 267.514,A -85,B 0,C 180,E1 -9063.872,E2 -9063.872} C_VEL
LIN {X 0,Y 444.232,Z 273.802,A -85,B 0,C 180,E1 -9064.964,E2 -9064.964} C_VEL
LIN {X 0,Y 444.003,Z 280.079,A -85,B 0,C 180,E1 -9065.947,E2 -9065.947} C_VEL
LIN {X 0,Y 442.717,Z 297.184,A -85,B 0,C 180,E1 -9068.555,E2 -9068.555} C_VEL
LIN {X 0,Y 444.406,Z 307.724,A -85,B 0,C 180,E1 -9068.849,E2 -9068.849} C_VEL
LIN {X 0,Y 445.769,Z 316.914,A -85,B 0,C 180,E1 -9069.071,E2 -9069.071} C_VEL
LIN {X 0,Y 444.177,Z 432.052,A -85,B 0,C 180,E1 -9071.044,E2 -9071.044} C_VEL
LIN {X 0,Y 443.75,Z 446.482,A -85,B 0,C 180,E1 -9071.474,E2 -9071.474} C_VEL
LIN {X 0,Y 443.179,Z 459.827,A -85,B 0,C 180,E1 -9072.048,E2 -9072.048} C_VEL
LIN {X 0,Y 442.547,Z 472.89,A -85,B 0,C 180,E1 -9072.796,E2 -9072.796} C_VEL
LIN {X 0,Y 441.767,Z 485.563,A -85,B 0,C 180,E1 -9073.717,E2 -9073.717} C_VEL
LIN {X 0,Y 440.959,Z 498.306,A -85,B 0,C 180,E1 -9074.872,E2 -9074.872} C_VEL
LIN {X 0,Y 440.255,Z 509.617,A -85,B 0,C 180,E1 -9076.146,E2 -9076.146} C_VEL
LIN {X 0,Y 439.728,Z 519.98,A -85,B 0,C 180,E1 -9077.574,E2 -9077.574} C_VEL
LIN {X 0,Y 439.137,Z 529.402,A -85,B 0,C 180,E1 -9079.161,E2 -9079.161} C_VEL
LIN {X 0,Y 438.752,Z 537.182,A -85,B 0,C 180,E1 -9080.783,E2 -9080.783} C_VEL
LIN {X 0,Y 438.522,Z 542.556,A -85,B 0,C 180,E1 -9082.171,E2 -9082.171} C_VEL
LIN {X 0,Y 438.412,Z 547.228,A -85,B 0,C 180,E1 -9083.665,E2 -9083.665} C_VEL
LIN {X 0,Y 438.313,Z 551.319,A -85,B 0,C 180,E1 -9085.402,E2 -9085.402} C_VEL
LIN {X 0,Y 438.336,Z 554.204,A -85,B 0,C 180,E1 -9087.243,E2 -9087.243} C_VEL
LIN {X 0,Y 438.25,Z 555.656,A -85,B 0,C 180,E1 -9089.081,E2 -9089.081} C_VEL
LIN {X 0,Y 438.25,Z 555.699,A -85,B 0,C 180,E1 -9090.919,E2 -9090.919} C_VEL
LIN {X 0,Y 438.336,Z 554.322,A -85,B 0,C 180,E1 -9092.757,E2 -9092.757} C_VEL
LIN {X 0,Y 438.316,Z 551.509,A -85,B 0,C 180,E1 -9094.598,E2 -9094.598} C_VEL
LIN {X 0,Y 438.421,Z 547.197,A -85,B 0,C 180,E1 -9096.443,E2 -9096.443} C_VEL
LIN {X 0,Y 438.602,Z 541.261,A -85,B 0,C 180,E1 -9098.292,E2 -9098.292} C_VEL
LIN {X 0,Y 438.885,Z 534.559,A -85,B 0,C 180,E1 -9099.912,E2 -9099.912} C_VEL
LIN {X 0,Y 439.404,Z 526.204,A -85,B 0,C 180,E1 -9101.533,E2 -9101.533} C_VEL
LIN {X 0,Y 439.933,Z 517.107,A -85,B 0,C 180,E1 -9102.971,E2 -9102.971} C_VEL
LIN {X 0,Y 440.573,Z 506.804,A -85,B 0,C 180,E1 -9104.315,E2 -9104.315} C_VEL
LIN {X 0,Y 441.265,Z 496.076,A -85,B 0,C 180,E1 -9105.472,E2 -9105.472} C_VEL
LIN {X 0,Y 442.077,Z 484.366,A -85,B 0,C 180,E1 -9106.509,E2 -9106.509} C_VEL
LIN {X 0,Y 442.852,Z 471.472,A -85,B 0,C 180,E1 -9107.43,E2 -9107.43} C_VEL
LIN {X 0,Y 443.576,Z 457.973,A -85,B 0,C 180,E1 -9108.18,E2 -9108.18} C_VEL
LIN {X 0,Y 444.117,Z 444.985,A -85,B 0,C 180,E1 -9108.72,E2 -9108.72} C_VEL
LIN {X 0,Y 444.601,Z 430.901,A -85,B 0,C 180,E1 -9109.117,E2 -9109.117} C_VEL
LIN {X 0,Y 446.089,Z 316.13,A -85,B 0,C 180,E1 -9111.096,E2 -9111.096} C_VEL
LIN {X 0,Y 442.98,Z 297.255,A -85,B 0,C 180,E1 -9111.615,E2 -9111.615} C_VEL
LIN {X 0,Y 444.414,Z 278.339,A -85,B 0,C 180,E1 -9114.526,E2 -9114.526} C_VEL
LIN {X 0,Y 444.583,Z 275.233,A -85,B 0,C 180,E1 -9115.015,E2 -9115.015} C_VEL
LIN {X 0,Y 441.764,Z 262.447,A -85,B 0,C 180,E1 -9117.291,E2 -9117.291} C_VEL
LIN {X 0,Y 439.44,Z 253.478,A -85,B 0,C 180,E1 -9118.998,E2 -9118.998} C_VEL
LIN {X 0,Y 439.368,Z 253.362,A -85,B 0,C 180,E1 -9122.03,E2 -9122.03} C_VEL
LIN {X 0,Y 439.392,Z 253.364,A -85,B 0,C 180,E1 -9125.34,E2 -9125.34} C_VEL
LIN {X 0,Y 439.375,Z 253.379,A -85,B 0,C 180,E1 -9128.595,E2 -9128.595} C_VEL
LIN {X 0,Y 439.392,Z 253.372,A -85,B 0,C 180,E1 -9131.257,E2 -9131.257} C_VEL
LIN {X 0,Y 439.405,Z 253.369,A -85,B 0,C 180,E1 -9134.728,E2 -9134.728} C_VEL
LIN {X 0,Y 439.391,Z 253.375,A -85,B 0,C 180,E1 -9137.795,E2 -9137.795} C_VEL
LIN {X 0,Y 439.432,Z 253.37,A -85,B 0,C 180,E1 -9140.228,E2 -9140.228} C_VEL
LIN {X 0,Y 439.372,Z 253.368,A -85,B 0,C 180,E1 -9143.713,E2 -9143.713} C_VEL
LIN {X 0,Y 439.367,Z 253.378,A -85,B 0,C 180,E1 -9147.054,E2 -9147.054} C_VEL
LIN {X 0,Y 439.39,Z 253.361,A -85,B 0,C 180,E1 -9150.275,E2 -9150.275} C_VEL
LIN {X 0,Y 439.424,Z 253.371,A -85,B 0,C 180,E1 -9153.396,E2 -9153.396} C_VEL
LIN {X 0,Y 439.381,Z 253.377,A -85,B 0,C 180,E1 -9156.429,E2 -9156.429} C_VEL
LIN {X 0,Y 439.382,Z 253.375,A -85,B 0,C 180,E1 -9159.397,E2 -9159.397} C_VEL
LIN {X 0,Y 439.425,Z 253.37,A -85,B 0,C 180,E1 -9162.31,E2 -9162.31} C_VEL
LIN {X 0,Y 439.441,Z 253.367,A -85,B 0,C 180,E1 -9165.174,E2 -9165.174} C_VEL
LIN {X 0,Y 439.477,Z 253.362,A -85,B 0,C 180,E1 -9168.001,E2 -9168.001} C_VEL
LIN {X 0,Y 439.541,Z 253.356,A -85,B 0,C 180,E1 -9171.726,E2 -9171.726} C_VEL
LIN {X 0,Y 439.615,Z 253.346,A -85,B 0,C 180,E1 -9174.496,E2 -9174.496} C_VEL
LIN {X 0,Y 439.629,Z 253.344,A -85,B 0,C 180,E1 -9178.168,E2 -9178.168} C_VEL
LIN {X 0,Y 439.757,Z 253.331,A -85,B 0,C 180,E1 -9180,E2 -9180} C_VEL
LIN {X 0,Y 439.65,Z 253.336,A -85,B 0,C 180,E1 -9182.749,E2 -9182.749} C_VEL
LIN {X 0,Y 439.612,Z 253.342,A -85,B 0,C 180,E1 -9186.426,E2 -9186.426} C_VEL
LIN {X 0,Y 439.494,Z 253.366,A -85,B 0,C 180,E1 -9189.202,E2 -9189.202} C_VEL
LIN {X 0,Y 439.46,Z 253.366,A -85,B 0,C 180,E1 -9192.938,E2 -9192.938} C_VEL
LIN {X 0,Y 439.442,Z 253.364,A -85,B 0,C 180,E1 -9196.349,E2 -9196.349} C_VEL
LIN {X 0,Y 439.398,Z 253.371,A -85,B 0,C 180,E1 -9199.627,E2 -9199.627} C_VEL
LIN {X 0,Y 439.36,Z 253.38,A -85,B 0,C 180,E1 -9202.576,E2 -9202.576} C_VEL
LIN {X 0,Y 439.401,Z 253.376,A -85,B 0,C 180,E1 -9205.586,E2 -9205.586} C_VEL
LIN {X 0,Y 439.414,Z 253.361,A -85,B 0,C 180,E1 -9208.674,E2 -9208.674} C_VEL
LIN {X 0,Y 439.368,Z 253.378,A -85,B 0,C 180,E1 -9212.031,E2 -9212.031} C_VEL
LIN {X 0,Y 439.394,Z 253.367,A -85,B 0,C 180,E1 -9215.341,E2 -9215.341} C_VEL
LIN {X 0,Y 439.381,Z 253.38,A -85,B 0,C 180,E1 -9218.596,E2 -9218.596} C_VEL
LIN {X 0,Y 439.387,Z 253.378,A -85,B 0,C 180,E1 -9221.258,E2 -9221.258} C_VEL
LIN {X 0,Y 439.401,Z 253.371,A -85,B 0,C 180,E1 -9224.73,E2 -9224.73} C_VEL
LIN {X 0,Y 439.398,Z 253.369,A -85,B 0,C 180,E1 -9227.797,E2 -9227.797} C_VEL
LIN {X 0,Y 439.437,Z 253.366,A -85,B 0,C 180,E1 -9230.229,E2 -9230.229} C_VEL
LIN {X 0,Y 439.374,Z 253.38,A -85,B 0,C 180,E1 -9233.714,E2 -9233.714} C_VEL
LIN {X 0,Y 439.373,Z 253.372,A -85,B 0,C 180,E1 -9237.055,E2 -9237.055} C_VEL
LIN {X 0,Y 439.413,Z 253.601,A -85,B 0,C 180,E1 -9238.48,E2 -9238.48} C_VEL
LIN {X 0,Y 442.505,Z 266.463,A -85,B 0,C 180,E1 -9241.112,E2 -9241.112} C_VEL
LIN {X 0,Y 443.856,Z 273.373,A -85,B 0,C 180,E1 -9242.463,E2 -9242.463} C_VEL
LIN {X 0,Y 443.091,Z 286.08,A -85,B 0,C 180,E1 -9244.703,E2 -9244.703} C_VEL
LIN {X 0,Y 442.057,Z 301.462,A -85,B 0,C 180,E1 -9247.366,E2 -9247.366} C_VEL
LIN {X 0,Y 441.449,Z 313.572,A -85,B 0,C 180,E1 -9249.391,E2 -9249.391} C_VEL
LIN {X 0,Y 445.259,Z 334.762,A -85,B 0,C 180,E1 -9249.932,E2 -9249.932} C_VEL
LIN {X 0,Y 444.551,Z 426.198,A -85,B 0,C 180,E1 -9251.359,E2 -9251.359} C_VEL
LIN {X 0,Y 444.115,Z 439.519,A -85,B 0,C 180,E1 -9251.753,E2 -9251.753} C_VEL
LIN {X 0,Y 444.037,Z 443.023,A -85,B 0,C 180,E1 -9251.89,E2 -9251.89} C_VEL
LIN {X 0,Y 443.188,Z 448.657,A -85,B 0,C 180,E1 -9252.116,E2 -9252.116} C_VEL
LIN {X 0,Y 438.601,Z 461.105,A -85,B 0,C 180,E1 -9252.655,E2 -9252.655} C_VEL
LIN {X 0,Y 436.267,Z 467.965,A -85,B 0,C 180,E1 -9253.064,E2 -9253.064} C_VEL
LIN {X 0,Y 435.689,Z 471.302,A -85,B 0,C 180,E1 -9253.317,E2 -9253.317} C_VEL
LIN {X 0,Y 434.808,Z 481.929,A -85,B 0,C 180,E1 -9254.292,E2 -9254.292} C_VEL
LIN {X 0,Y 434.167,Z 490.241,A -85,B 0,C 180,E1 -9255.23,E2 -9255.23} C_VEL
LIN {X 0,Y 433.406,Z 499.208,A -85,B 0,C 180,E1 -9256.449,E2 -9256.449} C_VEL
LIN {X 0,Y 432.833,Z 507.336,A -85,B 0,C 180,E1 -9257.814,E2 -9257.814} C_VEL
LIN {X 0,Y 432.231,Z 514.106,A -85,B 0,C 180,E1 -9259.223,E2 -9259.223} C_VEL
LIN {X 0,Y 431.854,Z 519.542,A -85,B 0,C 180,E1 -9260.634,E2 -9260.634} C_VEL
LIN {X 0,Y 431.614,Z 523.834,A -85,B 0,C 180,E1 -9262.044,E2 -9262.044} C_VEL
LIN {X 0,Y 431.374,Z 527.439,A -85,B 0,C 180,E1 -9263.632,E2 -9263.632} C_VEL
LIN {X 0,Y 431.25,Z 529.985,A -85,B 0,C 180,E1 -9265.326,E2 -9265.326} C_VEL
LIN {X 0,Y 431.274,Z 531.365,A -85,B 0,C 180,E1 -9267.198,E2 -9267.198} C_VEL
LIN {X 0,Y 431.173,Z 531.218,A -85,B 0,C 180,E1 -9269.066,E2 -9269.066} C_VEL
LIN {X 0,Y 431.206,Z 529.621,A -85,B 0,C 180,E1 -9270.934,E2 -9270.934} C_VEL
LIN {X 0,Y 431.293,Z 528.255,A -85,B 0,C 180,E1 -9271.868,E2 -9271.868} C_VEL
LIN {X 0,Y 431.622,Z 524.25,A -85,B 0,C 180,E1 -9273.734,E2 -9273.734} C_VEL
LIN {X 0,Y 431.801,Z 520.107,A -85,B 0,C 180,E1 -9275.136,E2 -9275.136} C_VEL
LIN {X 0,Y 432.174,Z 513.73,A -85,B 0,C 180,E1 -9276.802,E2 -9276.802} C_VEL
LIN {X 0,Y 432.68,Z 507.194,A -85,B 0,C 180,E1 -9278.147,E2 -9278.147} C_VEL
LIN {X 0,Y 433.216,Z 500.162,A -85,B 0,C 180,E1 -9279.336,E2 -9279.336} C_VEL
LIN {X 0,Y 433.876,Z 491.857,A -85,B 0,C 180,E1 -9280.499,E2 -9280.499} C_VEL
LIN {X 0,Y 434.623,Z 481.64,A -85,B 0,C 180,E1 -9281.661,E2 -9281.661} C_VEL
LIN {X 0,Y 435.345,Z 471.559,A -85,B 0,C 180,E1 -9282.588,E2 -9282.588} C_VEL
LIN {X 0,Y 435.908,Z 462.319,A -85,B 0,C 180,E1 -9283.282,E2 -9283.282} C_VEL
LIN {X 0,Y 436.514,Z 450.614,A -85,B 0,C 180,E1 -9283.975,E2 -9283.975} C_VEL
LIN {X 0,Y 437.117,Z 437.223,A -85,B 0,C 180,E1 -9284.549,E2 -9284.549} C_VEL
LIN {X 0,Y 437.432,Z 424.744,A -85,B 0,C 180,E1 -9284.896,E2 -9284.896} C_VEL
LIN {X 0,Y 438.146,Z 335.527,A -85,B 0,C 180,E1 -9286.291,E2 -9286.291} C_VEL
LIN {X 0,Y 434.385,Z 313.386,A -85,B 0,C 180,E1 -9286.84,E2 -9286.84} C_VEL
LIN {X 0,Y 435.424,Z 294.839,A -85,B 0,C 180,E1 -9290.011,E2 -9290.011} C_VEL
LIN {X 0,Y 436.743,Z 275.165,A -85,B 0,C 180,E1 -9293.473,E2 -9293.473} C_VEL
LIN {X 0,Y 435.875,Z 269.662,A -85,B 0,C 180,E1 -9294.531,E2 -9294.531} C_VEL
LIN {X 0,Y 432.46,Z 254.535,A -85,B 0,C 180,E1 -9297.591,E2 -9297.591} C_VEL
LIN {X 0,Y 432.389,Z 254.253,A -85,B 0,C 180,E1 -9298.122,E2 -9298.122} C_VEL
LIN {X 0,Y 432.323,Z 254.259,A -85,B 0,C 180,E1 -9301.345,E2 -9301.345} C_VEL
LIN {X 0,Y 432.341,Z 254.244,A -85,B 0,C 180,E1 -9304.676,E2 -9304.676} C_VEL
LIN {X 0,Y 432.339,Z 254.252,A -85,B 0,C 180,E1 -9308.149,E2 -9308.149} C_VEL
LIN {X 0,Y 432.334,Z 254.253,A -85,B 0,C 180,E1 -9311.601,E2 -9311.601} C_VEL
LIN {X 0,Y 432.34,Z 254.251,A -85,B 0,C 180,E1 -9314.345,E2 -9314.345} C_VEL
LIN {X 0,Y 432.319,Z 254.258,A -85,B 0,C 180,E1 -9317.015,E2 -9317.015} C_VEL
LIN {X 0,Y 432.331,Z 254.241,A -85,B 0,C 180,E1 -9319.82,E2 -9319.82} C_VEL
LIN {X 0,Y 432.313,Z 254.262,A -85,B 0,C 180,E1 -9323.022,E2 -9323.022} C_VEL
LIN {X 0,Y 432.356,Z 254.235,A -85,B 0,C 180,E1 -9325.996,E2 -9325.996} C_VEL
LIN {X 0,Y 432.391,Z 254.247,A -85,B 0,C 180,E1 -9329.743,E2 -9329.743} C_VEL
LIN {X 0,Y 432.395,Z 254.248,A -85,B 0,C 180,E1 -9333.372,E2 -9333.372} C_VEL
LIN {X 0,Y 432.366,Z 254.243,A -85,B 0,C 180,E1 -9336.023,E2 -9336.023} C_VEL
LIN {X 0,Y 432.344,Z 254.253,A -85,B 0,C 180,E1 -9339.045,E2 -9339.045} C_VEL
LIN {X 0,Y 432.372,Z 254.248,A -85,B 0,C 180,E1 -9342.011,E2 -9342.011} C_VEL
LIN {X 0,Y 432.39,Z 254.244,A -85,B 0,C 180,E1 -9344.926,E2 -9344.926} C_VEL
LIN {X 0,Y 432.453,Z 254.239,A -85,B 0,C 180,E1 -9347.803,E2 -9347.803} C_VEL
LIN {X 0,Y 432.485,Z 254.233,A -85,B 0,C 180,E1 -9351.59,E2 -9351.59} C_VEL
LIN {X 0,Y 432.591,Z 254.223,A -85,B 0,C 180,E1 -9354.406,E2 -9354.406} C_VEL
LIN {X 0,Y 432.599,Z 254.223,A -85,B 0,C 180,E1 -9358.138,E2 -9358.138} C_VEL
LIN {X 0,Y 432.726,Z 254.204,A -85,B 0,C 180,E1 -9360,E2 -9360} C_VEL
LIN {X 0,Y 432.598,Z 254.223,A -85,B 0,C 180,E1 -9362.793,E2 -9362.793} C_VEL
LIN {X 0,Y 432.566,Z 254.224,A -85,B 0,C 180,E1 -9366.53,E2 -9366.53} C_VEL
LIN {X 0,Y 432.436,Z 254.24,A -85,B 0,C 180,E1 -9369.353,E2 -9369.353} C_VEL
LIN {X 0,Y 432.424,Z 254.244,A -85,B 0,C 180,E1 -9372.803,E2 -9372.803} C_VEL
LIN {X 0,Y 432.405,Z 254.245,A -85,B 0,C 180,E1 -9376.479,E2 -9376.479} C_VEL
LIN {X 0,Y 432.332,Z 254.255,A -85,B 0,C 180,E1 -9379.961,E2 -9379.961} C_VEL
LIN {X 0,Y 432.313,Z 254.256,A -85,B 0,C 180,E1 -9382.964,E2 -9382.964} C_VEL
LIN {X 0,Y 432.358,Z 254.254,A -85,B 0,C 180,E1 -9386.033,E2 -9386.033} C_VEL
LIN {X 0,Y 432.346,Z 254.245,A -85,B 0,C 180,E1 -9389.187,E2 -9389.187} C_VEL
LIN {X 0,Y 432.32,Z 254.256,A -85,B 0,C 180,E1 -9392.294,E2 -9392.294} C_VEL
LIN {X 0,Y 432.335,Z 254.253,A -85,B 0,C 180,E1 -9394.677,E2 -9394.677} C_VEL
LIN {X 0,Y 432.342,Z 254.252,A -85,B 0,C 180,E1 -9398.149,E2 -9398.149} C_VEL
LIN {X 0,Y 432.328,Z 254.251,A -85,B 0,C 180,E1 -9401.602,E2 -9401.602} C_VEL
LIN {X 0,Y 432.332,Z 254.256,A -85,B 0,C 180,E1 -9404.347,E2 -9404.347} C_VEL
LIN {X 0,Y 432.316,Z 254.237,A -85,B 0,C 180,E1 -9407.016,E2 -9407.016} C_VEL
LIN {X 0,Y 432.337,Z 254.241,A -85,B 0,C 180,E1 -9409.82,E2 -9409.82} C_VEL
LIN {X 0,Y 432.303,Z 254.249,A -85,B 0,C 180,E1 -9413.023,E2 -9413.023} C_VEL
LIN {X 0,Y 432.357,Z 254.255,A -85,B 0,C 180,E1 -9415.997,E2 -9415.997} C_VEL
LIN {X 0,Y 432.346,Z 254.248,A -85,B 0,C 180,E1 -9419.49,E2 -9419.49} C_VEL
LIN {X 0,Y 432.425,Z 254.43,A -85,B 0,C 180,E1 -9420.994,E2 -9420.994} C_VEL
LIN {X 0,Y 435.947,Z 268.997,A -85,B 0,C 180,E1 -9423.684,E2 -9423.684} C_VEL
LIN {X 0,Y 437.498,Z 276.927,A -85,B 0,C 180,E1 -9425.072,E2 -9425.072} C_VEL
LIN {X 0,Y 435.88,Z 297.234,A -85,B 0,C 180,E1 -9428.233,E2 -9428.233} C_VEL
LIN {X 0,Y 436.658,Z 302.512,A -85,B 0,C 180,E1 -9428.405,E2 -9428.405} C_VEL
LIN {X 0,Y 439.051,Z 317.619,A -85,B 0,C 180,E1 -9428.785,E2 -9428.785} C_VEL
LIN {X 0,Y 437.42,Z 431.797,A -85,B 0,C 180,E1 -9430.77,E2 -9430.77} C_VEL
LIN {X 0,Y 436.943,Z 446.284,A -85,B 0,C 180,E1 -9431.205,E2 -9431.205} C_VEL
LIN {X 0,Y 436.328,Z 460.225,A -85,B 0,C 180,E1 -9431.817,E2 -9431.817} C_VEL
LIN {X 0,Y 435.618,Z 474.064,A -85,B 0,C 180,E1 -9432.635,E2 -9432.635} C_VEL
LIN {X 0,Y 434.805,Z 486.492,A -85,B 0,C 180,E1 -9433.569,E2 -9433.569} C_VEL
LIN {X 0,Y 434.01,Z 497.862,A -85,B 0,C 180,E1 -9434.624,E2 -9434.624} C_VEL
LIN {X 0,Y 433.302,Z 509.243,A -85,B 0,C 180,E1 -9435.919,E2 -9435.919} C_VEL
LIN {X 0,Y 432.795,Z 518.258,A -85,B 0,C 180,E1 -9437.155,E2 -9437.155} C_VEL
LIN {X 0,Y 432.281,Z 526.572,A -85,B 0,C 180,E1 -9438.512,E2 -9438.512} C_VEL
LIN {X 0,Y 431.762,Z 534.83,A -85,B 0,C 180,E1 -9440.159,E2 -9440.159} C_VEL
LIN {X 0,Y 431.513,Z 540.635,A -85,B 0,C 180,E1 -9441.571,E2 -9441.571} C_VEL
LIN {X 0,Y 431.335,Z 546.685,A -85,B 0,C 180,E1 -9443.451,E2 -9443.451} C_VEL
LIN {X 0,Y 431.237,Z 551.09,A -85,B 0,C 180,E1 -9445.326,E2 -9445.326} C_VEL
LIN {X 0,Y 431.231,Z 553.989,A -85,B 0,C 180,E1 -9447.198,E2 -9447.198} C_VEL
LIN {X 0,Y 431.166,Z 555.452,A -85,B 0,C 180,E1 -9449.066,E2 -9449.066} C_VEL
LIN {X 0,Y 431.166,Z 555.504,A -85,B 0,C 180,E1 -9450.934,E2 -9450.934} C_VEL
LIN {X 0,Y 431.231,Z 554.133,A -85,B 0,C 180,E1 -9452.802,E2 -9452.802} C_VEL
LIN {X 0,Y 431.241,Z 551.323,A -85,B 0,C 180,E1 -9454.674,E2 -9454.674} C_VEL
LIN {X 0,Y 431.335,Z 547.012,A -85,B 0,C 180,E1 -9456.549,E2 -9456.549} C_VEL
LIN {X 0,Y 431.557,Z 541.078,A -85,B 0,C 180,E1 -9458.428,E2 -9458.428} C_VEL
LIN {X 0,Y 431.842,Z 534.374,A -85,B 0,C 180,E1 -9460.076,E2 -9460.076} C_VEL
LIN {X 0,Y 432.393,Z 526.016,A -85,B 0,C 180,E1 -9461.722,E2 -9461.722} C_VEL
LIN {X 0,Y 432.942,Z 517.248,A -85,B 0,C 180,E1 -9463.136,E2 -9463.136} C_VEL
LIN {X 0,Y 433.64,Z 506.605,A -85,B 0,C 180,E1 -9464.549,E2 -9464.549} C_VEL
LIN {X 0,Y 434.403,Z 495.867,A -85,B 0,C 180,E1 -9465.723,E2 -9465.723} C_VEL
LIN {X 0,Y 435.229,Z 484.142,A -85,B 0,C 180,E1 -9466.776,E2 -9466.776} C_VEL
LIN {X 0,Y 436.06,Z 471.227,A -85,B 0,C 180,E1 -9467.71,E2 -9467.71} C_VEL
LIN {X 0,Y 436.794,Z 457.609,A -85,B 0,C 180,E1 -9468.477,E2 -9468.477} C_VEL
LIN {X 0,Y 437.412,Z 443.749,A -85,B 0,C 180,E1 -9469.048,E2 -9469.048} C_VEL
LIN {X 0,Y 437.899,Z 430.322,A -85,B 0,C 180,E1 -9469.422,E2 -9469.422} C_VEL
LIN {X 0,Y 439.442,Z 317.25,A -85,B 0,C 180,E1 -9471.4,E2 -9471.4} C_VEL
LIN {X 0,Y 436.224,Z 297.791,A -85,B 0,C 180,E1 -9471.924,E2 -9471.924} C_VEL
LIN {X 0,Y 436.7,Z 291.13,A -85,B 0,C 180,E1 -9472.92,E2 -9472.92} C_VEL
LIN {X 0,Y 437.787,Z 276.871,A -85,B 0,C 180,E1 -9475.177,E2 -9475.177} C_VEL
LIN {X 0,Y 434.849,Z 263.827,A -85,B 0,C 180,E1 -9477.547,E2 -9477.547} C_VEL
LIN {X 0,Y 432.371,Z 254.366,A -85,B 0,C 180,E1 -9479.385,E2 -9479.385} C_VEL
LIN {X 0,Y 432.321,Z 254.241,A -85,B 0,C 180,E1 -9482.443,E2 -9482.443} C_VEL
LIN {X 0,Y 432.342,Z 254.236,A -85,B 0,C 180,E1 -9485.631,E2 -9485.631} C_VEL
LIN {X 0,Y 432.343,Z 254.255,A -85,B 0,C 180,E1 -9489.343,E2 -9489.343} C_VEL
LIN {X 0,Y 432.367,Z 254.249,A -85,B 0,C 180,E1 -9491.792,E2 -9491.792} C_VEL
LIN {X 0,Y 432.375,Z 254.244,A -85,B 0,C 180,E1 -9494.341,E2 -9494.341} C_VEL
LIN {X 0,Y 432.329,Z 254.249,A -85,B 0,C 180,E1 -9498.203,E2 -9498.203} C_VEL
LIN {X 0,Y 432.348,Z 254.253,A -85,B 0,C 180,E1 -9501.283,E2 -9501.283} C_VEL
LIN {X 0,Y 432.341,Z 254.244,A -85,B 0,C 180,E1 -9504.368,E2 -9504.368} C_VEL
LIN {X 0,Y 432.318,Z 254.258,A -85,B 0,C 180,E1 -9507.557,E2 -9507.557} C_VEL
LIN {X 0,Y 432.389,Z 254.234,A -85,B 0,C 180,E1 -9509.744,E2 -9509.744} C_VEL
LIN {X 0,Y 432.394,Z 254.247,A -85,B 0,C 180,E1 -9513.372,E2 -9513.372} C_VEL
LIN {X 0,Y 432.366,Z 254.251,A -85,B 0,C 180,E1 -9516.023,E2 -9516.023} C_VEL
LIN {X 0,Y 432.344,Z 254.25,A -85,B 0,C 180,E1 -9519.046,E2 -9519.046} C_VEL
LIN {X 0,Y 432.372,Z 254.252,A -85,B 0,C 180,E1 -9522.011,E2 -9522.011} C_VEL
LIN {X 0,Y 432.389,Z 254.245,A -85,B 0,C 180,E1 -9524.926,E2 -9524.926} C_VEL
LIN {X 0,Y 432.452,Z 254.237,A -85,B 0,C 180,E1 -9527.804,E2 -9527.804} C_VEL
LIN {X 0,Y 432.485,Z 254.237,A -85,B 0,C 180,E1 -9531.59,E2 -9531.59} C_VEL
LIN {X 0,Y 432.591,Z 254.222,A -85,B 0,C 180,E1 -9534.406,E2 -9534.406} C_VEL
LIN {X 0,Y 432.599,Z 254.219,A -85,B 0,C 180,E1 -9538.138,E2 -9538.138} C_VEL
LIN {X 0,Y 432.727,Z 254.206,A -85,B 0,C 180,E1 -9540,E2 -9540} C_VEL
LIN {X 0,Y 432.6,Z 254.215,A -85,B 0,C 180,E1 -9542.794,E2 -9542.794} C_VEL
LIN {X 0,Y 432.567,Z 254.22,A -85,B 0,C 180,E1 -9546.531,E2 -9546.531} C_VEL
LIN {X 0,Y 432.437,Z 254.247,A -85,B 0,C 180,E1 -9549.354,E2 -9549.354} C_VEL
LIN {X 0,Y 432.425,Z 254.241,A -85,B 0,C 180,E1 -9552.804,E2 -9552.804} C_VEL
LIN {X 0,Y 432.407,Z 254.24,A -85,B 0,C 180,E1 -9556.48,E2 -9556.48} C_VEL
LIN {X 0,Y 432.333,Z 254.249,A -85,B 0,C 180,E1 -9559.961,E2 -9559.961} C_VEL
LIN {X 0,Y 432.315,Z 254.26,A -85,B 0,C 180,E1 -9562.965,E2 -9562.965} C_VEL
LIN {X 0,Y 432.36,Z 254.251,A -85,B 0,C 180,E1 -9566.033,E2 -9566.033} C_VEL
LIN {X 0,Y 432.339,Z 254.24,A -85,B 0,C 180,E1 -9569.188,E2 -9569.188} C_VEL
LIN {X 0,Y 432.32,Z 254.258,A -85,B 0,C 180,E1 -9572.444,E2 -9572.444} C_VEL
LIN {X 0,Y 432.343,Z 254.246,A -85,B 0,C 180,E1 -9575.633,E2 -9575.633} C_VEL
LIN {X 0,Y 432.343,Z 254.253,A -85,B 0,C 180,E1 -9578.716,E2 -9578.716} C_VEL
LIN {X 0,Y 432.332,Z 254.255,A -85,B 0,C 180,E1 -9581.798,E2 -9581.798} C_VEL
LIN {X 0,Y 432.333,Z 254.248,A -85,B 0,C 180,E1 -9584.348,E2 -9584.348} C_VEL
LIN {X 0,Y 432.325,Z 254.253,A -85,B 0,C 180,E1 -9587.016,E2 -9587.016} C_VEL
LIN {X 0,Y 432.342,Z 254.254,A -85,B 0,C 180,E1 -9589.82,E2 -9589.82} C_VEL
LIN {X 0,Y 432.307,Z 254.247,A -85,B 0,C 180,E1 -9593.023,E2 -9593.023} C_VEL
LIN {X 0,Y 432.359,Z 254.236,A -85,B 0,C 180,E1 -9595.998,E2 -9595.998} C_VEL
LIN {X 0,Y 432.371,Z 254.403,A -85,B 0,C 180,E1 -9598.087,E2 -9598.087} C_VEL
LIN {X 0,Y 435.336,Z 266.698,A -85,B 0,C 180,E1 -9600.666,E2 -9600.666} C_VEL
LIN {X 0,Y 437.045,Z 275.35,A -85,B 0,C 180,E1 -9602.388,E2 -9602.388} C_VEL
LIN {X 0,Y 436.081,Z 289.032,A -85,B 0,C 180,E1 -9604.828,E2 -9604.828} C_VEL
LIN {X 0,Y 435.058,Z 303.923,A -85,B 0,C 180,E1 -9607.44,E2 -9607.44} C_VEL
LIN {X 0,Y 434.578,Z 313.298,A -85,B 0,C 180,E1 -9609.035,E2 -9609.035} C_VEL
LIN {X 0,Y 438.684,Z 336.249,A -85,B 0,C 180,E1 -9609.639,E2 -9609.639} C_VEL
LIN {X 0,Y 437.845,Z 426.337,A -85,B 0,C 180,E1 -9611.063,E2 -9611.063} C_VEL
LIN {X 0,Y 437.37,Z 439.451,A -85,B 0,C 180,E1 -9611.454,E2 -9611.454} C_VEL
LIN {X 0,Y 436.886,Z 452.753,A -85,B 0,C 180,E1 -9612.062,E2 -9612.062} C_VEL
LIN {X 0,Y 436.216,Z 464.292,A -85,B 0,C 180,E1 -9612.78,E2 -9612.78} C_VEL
LIN {X 0,Y 435.689,Z 471.302,A -85,B 0,C 180,E1 -9613.317,E2 -9613.317} C_VEL
LIN {X 0,Y 434.632,Z 476.305,A -85,B 0,C 180,E1 -9613.721,E2 -9613.721} C_VEL
LIN {X 0,Y 431.217,Z 484.16,A -85,B 0,C 180,E1 -9614.394,E2 -9614.394} C_VEL
LIN {X 0,Y 427.833,Z 491.499,A -85,B 0,C 180,E1 -9615.151,E2 -9615.151} C_VEL
LIN {X 0,Y 426.805,Z 495.667,A -85,B 0,C 180,E1 -9615.685,E2 -9615.685} C_VEL
LIN {X 0,Y 426.054,Z 504.163,A -85,B 0,C 180,E1 -9617.01,E2 -9617.01} C_VEL
LIN {X 0,Y 425.569,Z 511.039,A -85,B 0,C 180,E1 -9618.329,E2 -9618.329} C_VEL
LIN {X 0,Y 424.935,Z 518.004,A -85,B 0,C 180,E1 -9619.999,E2 -9619.999} C_VEL
LIN {X 0,Y 424.611,Z 522.668,A -85,B 0,C 180,E1 -9621.433,E2 -9621.433} C_VEL
LIN {X 0,Y 424.405,Z 526.27,A -85,B 0,C 180,E1 -9622.866,E2 -9622.866} C_VEL
LIN {X 0,Y 424.235,Z 528.91,A -85,B 0,C 180,E1 -9624.296,E2 -9624.296} C_VEL
LIN {X 0,Y 424.12,Z 531.044,A -85,B 0,C 180,E1 -9626.199,E2 -9626.199} C_VEL
LIN {X 0,Y 424.172,Z 531.557,A -85,B 0,C 180,E1 -9627.151,E2 -9627.151} C_VEL
LIN {X 0,Y 424.093,Z 531.427,A -85,B 0,C 180,E1 -9629.05,E2 -9629.05} C_VEL
LIN {X 0,Y 424.124,Z 529.846,A -85,B 0,C 180,E1 -9630.949,E2 -9630.949} C_VEL
LIN {X 0,Y 424.218,Z 528.494,A -85,B 0,C 180,E1 -9631.899,E2 -9631.899} C_VEL
LIN {X 0,Y 424.447,Z 525.68,A -85,B 0,C 180,E1 -9633.322,E2 -9633.322} C_VEL
LIN {X 0,Y 424.59,Z 521.899,A -85,B 0,C 180,E1 -9634.747,E2 -9634.747} C_VEL
LIN {X 0,Y 424.931,Z 517.045,A -85,B 0,C 180,E1 -9636.171,E2 -9636.171} C_VEL
LIN {X 0,Y 425.376,Z 510.977,A -85,B 0,C 180,E1 -9637.595,E2 -9637.595} C_VEL
LIN {X 0,Y 425.949,Z 503.45,A -85,B 0,C 180,E1 -9639.018,E2 -9639.018} C_VEL
LIN {X 0,Y 426.629,Z 495.785,A -85,B 0,C 180,E1 -9640.2,E2 -9640.2} C_VEL
LIN {X 0,Y 427.516,Z 485.406,A -85,B 0,C 180,E1 -9641.497,E2 -9641.497} C_VEL
LIN {X 0,Y 428.215,Z 474.873,A -85,B 0,C 180,E1 -9642.56,E2 -9642.56} C_VEL
LIN {X 0,Y 429.039,Z 463.036,A -85,B 0,C 180,E1 -9643.499,E2 -9643.499} C_VEL
LIN {X 0,Y 429.678,Z 451.504,A -85,B 0,C 180,E1 -9644.202,E2 -9644.202} C_VEL
LIN {X 0,Y 430.299,Z 438.401,A -85,B 0,C 180,E1 -9644.785,E2 -9644.785} C_VEL
LIN {X 0,Y 430.675,Z 425.583,A -85,B 0,C 180,E1 -9645.162,E2 -9645.162} C_VEL
LIN {X 0,Y 431.376,Z 336.184,A -85,B 0,C 180,E1 -9646.588,E2 -9646.588} C_VEL
LIN {X 0,Y 427.481,Z 313.274,A -85,B 0,C 180,E1 -9647.167,E2 -9647.167} C_VEL
LIN {X 0,Y 428.574,Z 295.031,A -85,B 0,C 180,E1 -9650.331,E2 -9650.331} C_VEL
LIN {X 0,Y 429.88,Z 276.103,A -85,B 0,C 180,E1 -9653.717,E2 -9653.717} C_VEL
LIN {X 0,Y 427.437,Z 264.236,A -85,B 0,C 180,E1 -9656.094,E2 -9656.094} C_VEL
LIN {X 0,Y 425.384,Z 255.192,A -85,B 0,C 180,E1 -9658.023,E2 -9658.023} C_VEL
LIN {X 0,Y 425.29,Z 255.129,A -85,B 0,C 180,E1 -9660.815,E2 -9660.815} C_VEL
LIN {X 0,Y 425.312,Z 255.114,A -85,B 0,C 180,E1 -9664.287,E2 -9664.287} C_VEL
LIN {X 0,Y 425.28,Z 255.131,A -85,B 0,C 180,E1 -9667.693,E2 -9667.693} C_VEL
LIN {X 0,Y 425.282,Z 255.131,A -85,B 0,C 180,E1 -9670.52,E2 -9670.52} C_VEL
LIN {X 0,Y 425.263,Z 255.138,A -85,B 0,C 180,E1 -9673.351,E2 -9673.351} C_VEL
LIN {X 0,Y 425.256,Z 255.134,A -85,B 0,C 180,E1 -9676.648,E2 -9676.648} C_VEL
LIN {X 0,Y 425.283,Z 255.118,A -85,B 0,C 180,E1 -9679.872,E2 -9679.872} C_VEL
LIN {X 0,Y 425.281,Z 255.132,A -85,B 0,C 180,E1 -9682.487,E2 -9682.487} C_VEL
LIN {X 0,Y 425.305,Z 255.113,A -85,B 0,C 180,E1 -9685.816,E2 -9685.816} C_VEL
LIN {X 0,Y 425.297,Z 255.135,A -85,B 0,C 180,E1 -9689.236,E2 -9689.236} C_VEL
LIN {X 0,Y 425.345,Z 255.121,A -85,B 0,C 180,E1 -9692.442,E2 -9692.442} C_VEL
LIN {X 0,Y 425.347,Z 255.118,A -85,B 0,C 180,E1 -9695.601,E2 -9695.601} C_VEL
LIN {X 0,Y 425.288,Z 255.137,A -85,B 0,C 180,E1 -9698.681,E2 -9698.681} C_VEL
LIN {X 0,Y 425.327,Z 255.125,A -85,B 0,C 180,E1 -9701.702,E2 -9701.702} C_VEL
LIN {X 0,Y 425.343,Z 255.123,A -85,B 0,C 180,E1 -9704.67,E2 -9704.67} C_VEL
LIN {X 0,Y 425.406,Z 255.117,A -85,B 0,C 180,E1 -9707.598,E2 -9707.598} C_VEL
LIN {X 0,Y 425.436,Z 255.111,A -85,B 0,C 180,E1 -9711.449,E2 -9711.449} C_VEL
LIN {X 0,Y 425.547,Z 255.101,A -85,B 0,C 180,E1 -9714.313,E2 -9714.313} C_VEL
LIN {X 0,Y 425.569,Z 255.099,A -85,B 0,C 180,E1 -9718.107,E2 -9718.107} C_VEL
LIN {X 0,Y 425.696,Z 255.08,A -85,B 0,C 180,E1 -9720,E2 -9720} C_VEL
LIN {X 0,Y 425.55,Z 255.101,A -85,B 0,C 180,E1 -9722.84,E2 -9722.84} C_VEL
LIN {X 0,Y 425.524,Z 255.102,A -85,B 0,C 180,E1 -9726.639,E2 -9726.639} C_VEL
LIN {X 0,Y 425.394,Z 255.117,A -85,B 0,C 180,E1 -9729.509,E2 -9729.509} C_VEL
LIN {X 0,Y 425.386,Z 255.12,A -85,B 0,C 180,E1 -9732.904,E2 -9732.904} C_VEL
LIN {X 0,Y 425.354,Z 255.124,A -85,B 0,C 180,E1 -9736.605,E2 -9736.605} C_VEL
LIN {X 0,Y 425.322,Z 255.128,A -85,B 0,C 180,E1 -9739.636,E2 -9739.636} C_VEL
LIN {X 0,Y 425.301,Z 255.13,A -85,B 0,C 180,E1 -9743.365,E2 -9743.365} C_VEL
LIN {X 0,Y 425.342,Z 255.125,A -85,B 0,C 180,E1 -9746.845,E2 -9746.845} C_VEL
LIN {X 0,Y 425.312,Z 255.116,A -85,B 0,C 180,E1 -9749.718,E2 -9749.718} C_VEL
LIN {X 0,Y 425.276,Z 255.133,A -85,B 0,C 180,E1 -9753.048,E2 -9753.048} C_VEL
LIN {X 0,Y 425.279,Z 255.125,A -85,B 0,C 180,E1 -9755.929,E2 -9755.929} C_VEL
LIN {X 0,Y 425.298,Z 255.131,A -85,B 0,C 180,E1 -9759.045,E2 -9759.045} C_VEL
LIN {X 0,Y 425.27,Z 255.129,A -85,B 0,C 180,E1 -9762.653,E2 -9762.653} C_VEL
LIN {X 0,Y 425.257,Z 255.126,A -85,B 0,C 180,E1 -9766.045,E2 -9766.045} C_VEL
LIN {X 0,Y 425.27,Z 255.104,A -85,B 0,C 180,E1 -9768.622,E2 -9768.622} C_VEL
LIN {X 0,Y 425.309,Z 255.131,A -85,B 0,C 180,E1 -9771.103,E2 -9771.103} C_VEL
LIN {X 0,Y 425.296,Z 255.112,A -85,B 0,C 180,E1 -9774.665,E2 -9774.665} C_VEL
LIN {X 0,Y 425.262,Z 255.12,A -85,B 0,C 180,E1 -9778.074,E2 -9778.074} C_VEL
LIN {X 0,Y 425.332,Z 255.281,A -85,B 0,C 180,E1 -9780.621,E2 -9780.621} C_VEL
LIN {X 0,Y 428.741,Z 268.908,A -85,B 0,C 180,E1 -9783.207,E2 -9783.207} C_VEL
LIN {X 0,Y 430.666,Z 278.329,A -85,B 0,C 180,E1 -9784.895,E2 -9784.895} C_VEL
LIN {X 0,Y 429.077,Z 297.549,A -85,B 0,C 180,E1 -9787.928,E2 -9787.928} C_VEL
LIN {X 0,Y 432.291,Z 317.846,A -85,B 0,C 180,E1 -9788.479,E2 -9788.479} C_VEL
LIN {X 0,Y 430.662,Z 431.531,A -85,B 0,C 180,E1 -9790.487,E2 -9790.487} C_VEL
LIN {X 0,Y 430.137,Z 446.087,A -85,B 0,C 180,E1 -9790.927,E2 -9790.927} C_VEL
LIN {X 0,Y 429.51,Z 460.349,A -85,B 0,C 180,E1 -9791.565,E2 -9791.565} C_VEL
LIN {X 0,Y 428.811,Z 473.464,A -85,B 0,C 180,E1 -9792.35,E2 -9792.35} C_VEL
LIN {X 0,Y 427.915,Z 485.98,A -85,B 0,C 180,E1 -9793.297,E2 -9793.297} C_VEL
LIN {X 0,Y 427.148,Z 497.42,A -85,B 0,C 180,E1 -9794.37,E2 -9794.37} C_VEL
LIN {X 0,Y 426.449,Z 506.928,A -85,B 0,C 180,E1 -9795.444,E2 -9795.444} C_VEL
LIN {X 0,Y 425.792,Z 517.419,A -85,B 0,C 180,E1 -9796.865,E2 -9796.865} C_VEL
LIN {X 0,Y 425.278,Z 526.26,A -85,B 0,C 180,E1 -9798.321,E2 -9798.321} C_VEL
LIN {X 0,Y 424.706,Z 534.546,A -85,B 0,C 180,E1 -9799.994,E2 -9799.994} C_VEL
LIN {X 0,Y 424.448,Z 540.371,A -85,B 0,C 180,E1 -9801.43,E2 -9801.43} C_VEL
LIN {X 0,Y 424.314,Z 545.089,A -85,B 0,C 180,E1 -9802.864,E2 -9802.864} C_VEL
LIN {X 0,Y 424.152,Z 549.935,A -85,B 0,C 180,E1 -9804.771,E2 -9804.771} C_VEL
LIN {X 0,Y 424.086,Z 552.499,A -85,B 0,C 180,E1 -9806.199,E2 -9806.199} C_VEL
LIN {X 0,Y 424.126,Z 554.687,A -85,B 0,C 180,E1 -9808.101,E2 -9808.101} C_VEL
LIN {X 0,Y 424.082,Z 555.456,A -85,B 0,C 180,E1 -9810,E2 -9810} C_VEL
LIN {X 0,Y 424.126,Z 554.807,A -85,B 0,C 180,E1 -9811.899,E2 -9811.899} C_VEL
LIN {X 0,Y 424.086,Z 552.723,A -85,B 0,C 180,E1 -9813.801,E2 -9813.801} C_VEL
LIN {X 0,Y 424.166,Z 551.14,A -85,B 0,C 180,E1 -9814.752,E2 -9814.752} C_VEL
LIN {X 0,Y 424.245,Z 546.83,A -85,B 0,C 180,E1 -9816.659,E2 -9816.659} C_VEL
LIN {X 0,Y 424.483,Z 540.897,A -85,B 0,C 180,E1 -9818.569,E2 -9818.569} C_VEL
LIN {X 0,Y 424.79,Z 534.193,A -85,B 0,C 180,E1 -9820.245,E2 -9820.245} C_VEL
LIN {X 0,Y 425.387,Z 525.832,A -85,B 0,C 180,E1 -9821.918,E2 -9821.918} C_VEL
LIN {X 0,Y 425.966,Z 517.061,A -85,B 0,C 180,E1 -9823.355,E2 -9823.355} C_VEL
LIN {X 0,Y 426.725,Z 506.413,A -85,B 0,C 180,E1 -9824.79,E2 -9824.79} C_VEL
LIN {X 0,Y 427.63,Z 494.481,A -85,B 0,C 180,E1 -9826.101,E2 -9826.101} C_VEL
LIN {X 0,Y 428.501,Z 482.493,A -85,B 0,C 180,E1 -9827.171,E2 -9827.171} C_VEL
LIN {X 0,Y 429.369,Z 469.164,A -85,B 0,C 180,E1 -9828.119,E2 -9828.119} C_VEL
LIN {X 0,Y 430.115,Z 455.651,A -85,B 0,C 180,E1 -9828.856,E2 -9828.856} C_VEL
LIN {X 0,Y 430.791,Z 441.58,A -85,B 0,C 180,E1 -9829.414,E2 -9829.414} C_VEL
LIN {X 0,Y 431.246,Z 426.872,A -85,B 0,C 180,E1 -9829.796,E2 -9829.796} C_VEL
LIN {X 0,Y 432.776,Z 317.47,A -85,B 0,C 180,E1 -9831.731,E2 -9831.731} C_VEL
LIN {X 0,Y 429.461,Z 297.584,A -85,B 0,C 180,E1 -9832.3,E2 -9832.3} C_VEL
LIN {X 0,Y 430.917,Z 280.055,A -85,B 0,C 180,E1 -9835.09,E2 -9835.09} C_VEL
LIN {X 0,Y 430.77,Z 277.405,A -85,B 0,C 180,E1 -9835.542,E2 -9835.542} C_VEL
LIN {X 0,Y 427.773,Z 264.584,A -85,B 0,C 180,E1 -9837.931,E2 -9837.931} C_VEL
LIN {X 0,Y 425.338,Z 255.226,A -85,B 0,C 180,E1 -9839.801,E2 -9839.801} C_VEL
LIN {X 0,Y 425.28,Z 255.125,A -85,B 0,C 180,E1 -9843.048,E2 -9843.048} C_VEL
LIN {X 0,Y 425.279,Z 255.112,A -85,B 0,C 180,E1 -9845.928,E2 -9845.928} C_VEL
LIN {X 0,Y 425.29,Z 255.134,A -85,B 0,C 180,E1 -9849.042,E2 -9849.042} C_VEL
LIN {X 0,Y 425.328,Z 255.13,A -85,B 0,C 180,E1 -9852.646,E2 -9852.646} C_VEL
LIN {X 0,Y 425.291,Z 255.128,A -85,B 0,C 180,E1 -9855.281,E2 -9855.281} C_VEL
LIN {X 0,Y 425.27,Z 255.125,A -85,B 0,C 180,E1 -9858.621,E2 -9858.621} C_VEL
LIN {X 0,Y 425.311,Z 255.13,A -85,B 0,C 180,E1 -9861.103,E2 -9861.103} C_VEL
LIN {X 0,Y 425.295,Z 255.123,A -85,B 0,C 180,E1 -9864.664,E2 -9864.664} C_VEL
LIN {X 0,Y 425.261,Z 255.134,A -85,B 0,C 180,E1 -9868.073,E2 -9868.073} C_VEL
LIN {X 0,Y 425.332,Z 255.115,A -85,B 0,C 180,E1 -9871.368,E2 -9871.368} C_VEL
LIN {X 0,Y 425.29,Z 255.13,A -85,B 0,C 180,E1 -9874.555,E2 -9874.555} C_VEL
LIN {X 0,Y 425.282,Z 255.136,A -85,B 0,C 180,E1 -9877.661,E2 -9877.661} C_VEL
LIN {X 0,Y 425.356,Z 255.122,A -85,B 0,C 180,E1 -9880.704,E2 -9880.704} C_VEL
LIN {X 0,Y 425.382,Z 255.118,A -85,B 0,C 180,E1 -9883.688,E2 -9883.688} C_VEL
LIN {X 0,Y 425.405,Z 255.116,A -85,B 0,C 180,E1 -9887.598,E2 -9887.598} C_VEL
LIN {X 0,Y 425.436,Z 255.117,A -85,B 0,C 180,E1 -9891.45,E2 -9891.45} C_VEL
LIN {X 0,Y 425.548,Z 255.1,A -85,B 0,C 180,E1 -9894.313,E2 -9894.313} C_VEL
LIN {X 0,Y 425.569,Z 255.095,A -85,B 0,C 180,E1 -9898.108,E2 -9898.108} C_VEL
LIN {X 0,Y 425.697,Z 255.082,A -85,B 0,C 180,E1 -9900,E2 -9900} C_VEL
LIN {X 0,Y 425.551,Z 255.093,A -85,B 0,C 180,E1 -9902.84,E2 -9902.84} C_VEL
LIN {X 0,Y 425.525,Z 255.097,A -85,B 0,C 180,E1 -9906.644,E2 -9906.644} C_VEL
LIN {X 0,Y 425.395,Z 255.122,A -85,B 0,C 180,E1 -9909.51,E2 -9909.51} C_VEL
LIN {X 0,Y 425.388,Z 255.118,A -85,B 0,C 180,E1 -9912.904,E2 -9912.904} C_VEL
LIN {X 0,Y 425.356,Z 255.119,A -85,B 0,C 180,E1 -9916.606,E2 -9916.606} C_VEL
LIN {X 0,Y 425.324,Z 255.124,A -85,B 0,C 180,E1 -9919.636,E2 -9919.636} C_VEL
LIN {X 0,Y 425.303,Z 255.129,A -85,B 0,C 180,E1 -9923.366,E2 -9923.366} C_VEL
LIN {X 0,Y 425.344,Z 255.127,A -85,B 0,C 180,E1 -9926.845,E2 -9926.845} C_VEL
LIN {X 0,Y 425.287,Z 255.122,A -85,B 0,C 180,E1 -9929.72,E2 -9929.72} C_VEL
LIN {X 0,Y 425.28,Z 255.134,A -85,B 0,C 180,E1 -9933.049,E2 -9933.049} C_VEL
LIN {X 0,Y 425.282,Z 255.126,A -85,B 0,C 180,E1 -9935.93,E2 -9935.93} C_VEL
LIN {X 0,Y 425.289,Z 255.126,A -85,B 0,C 180,E1 -9939.043,E2 -9939.043} C_VEL
LIN {X 0,Y 425.274,Z 255.138,A -85,B 0,C 180,E1 -9942.654,E2 -9942.654} C_VEL
LIN {X 0,Y 425.268,Z 255.137,A -85,B 0,C 180,E1 -9946.046,E2 -9946.046} C_VEL
LIN {X 0,Y 425.285,Z 255.133,A -85,B 0,C 180,E1 -9949.48,E2 -9949.48} C_VEL
LIN {X 0,Y 425.279,Z 255.113,A -85,B 0,C 180,E1 -9952.489,E2 -9952.489} C_VEL
LIN {X 0,Y 425.307,Z 255.114,A -85,B 0,C 180,E1 -9955.818,E2 -9955.818} C_VEL
LIN {X 0,Y 425.327,Z 255.35,A -85,B 0,C 180,E1 -9957.722,E2 -9957.722} C_VEL
LIN {X 0,Y 428.516,Z 268.509,A -85,B 0,C 180,E1 -9960.527,E2 -9960.527} C_VEL
LIN {X 0,Y 430.153,Z 276.44,A -85,B 0,C 180,E1 -9962.14,E2 -9962.14} C_VEL
LIN {X 0,Y 429.652,Z 285.482,A -85,B 0,C 180,E1 -9963.791,E2 -9963.791} C_VEL
LIN {X 0,Y 428.373,Z 302.404,A -85,B 0,C 180,E1 -9966.812,E2 -9966.812} C_VEL
LIN {X 0,Y 427.717,Z 313.234,A -85,B 0,C 180,E1 -9968.682,E2 -9968.682} C_VEL
LIN {X 0,Y 431.992,Z 336.794,A -85,B 0,C 180,E1 -9969.315,E2 -9969.315} C_VEL
LIN {X 0,Y 431.138,Z 426.475,A -85,B 0,C 180,E1 -9970.757,E2 -9970.757} C_VEL
LIN {X 0,Y 430.642,Z 440.083,A -85,B 0,C 180,E1 -9971.174,E2 -9971.174} C_VEL
LIN {X 0,Y 430.134,Z 453.06,A -85,B 0,C 180,E1 -9971.782,E2 -9971.782} C_VEL
LIN {X 0,Y 429.448,Z 464.402,A -85,B 0,C 180,E1 -9972.5,E2 -9972.5} C_VEL
LIN {X 0,Y 428.499,Z 475.981,A -85,B 0,C 180,E1 -9973.443,E2 -9973.443} C_VEL
LIN {X 0,Y 427.691,Z 486.385,A -85,B 0,C 180,E1 -9974.513,E2 -9974.513} C_VEL
LIN {X 0,Y 426.805,Z 495.667,A -85,B 0,C 180,E1 -9975.685,E2 -9975.685} C_VEL
LIN {X 0,Y 425.805,Z 499.737,A -85,B 0,C 180,E1 -9976.247,E2 -9976.247} C_VEL
LIN {X 0,Y 422.495,Z 505.967,A -85,B 0,C 180,E1 -9977.191,E2 -9977.191} C_VEL
LIN {X 0,Y 419.197,Z 511.531,A -85,B 0,C 180,E1 -9978.217,E2 -9978.217} C_VEL
LIN {X 0,Y 418.229,Z 514.558,A -85,B 0,C 180,E1 -9978.9,E2 -9978.9} C_VEL
LIN {X 0,Y 417.766,Z 519.841,A -85,B 0,C 180,E1 -9980.315,E2 -9980.315} C_VEL
LIN {X 0,Y 417.494,Z 524.15,A -85,B 0,C 180,E1 -9981.774,E2 -9981.774} C_VEL
LIN {X 0,Y 417.201,Z 528.224,A -85,B 0,C 180,E1 -9983.669,E2 -9983.669} C_VEL
LIN {X 0,Y 417.111,Z 530.34,A -85,B 0,C 180,E1 -9985.167,E2 -9985.167} C_VEL
LIN {X 0,Y 417.07,Z 531.748,A -85,B 0,C 180,E1 -9987.102,E2 -9987.102} C_VEL
LIN {X 0,Y 417.074,Z 531.877,A -85,B 0,C 180,E1 -9988.069,E2 -9988.069} C_VEL
LIN {X 0,Y 417.009,Z 531.034,A -85,B 0,C 180,E1 -9990,E2 -9990} C_VEL
LIN {X 0,Y 417.145,Z 528.731,A -85,B 0,C 180,E1 -9991.931,E2 -9991.931} C_VEL
LIN {X 0,Y 417.385,Z 525.931,A -85,B 0,C 180,E1 -9993.378,E2 -9993.378} C_VEL
LIN {X 0,Y 417.52,Z 522.172,A -85,B 0,C 180,E1 -9994.828,E2 -9994.828} C_VEL
LIN {X 0,Y 417.895,Z 517.341,A -85,B 0,C 180,E1 -9996.276,E2 -9996.276} C_VEL
LIN {X 0,Y 418.363,Z 511.301,A -85,B 0,C 180,E1 -9997.723,E2 -9997.723} C_VEL
LIN {X 0,Y 418.972,Z 503.821,A -85,B 0,C 180,E1 -9999.169,E2 -9999.169} C_VEL
LIN {X 0,Y 419.803,Z 494.461,A -85,B 0,C 180,E1 -10000.612,E2 -10000.612} C_VEL
LIN {X 0,Y 420.675,Z 484.832,A -85,B 0,C 180,E1 -10001.809,E2 -10001.809} C_VEL
LIN {X 0,Y 421.327,Z 475.421,A -85,B 0,C 180,E1 -10002.769,E2 -10002.769} C_VEL
LIN {X 0,Y 422.165,Z 463.74,A -85,B 0,C 180,E1 -10003.723,E2 -10003.723} C_VEL
LIN {X 0,Y 422.848,Z 452.384,A -85,B 0,C 180,E1 -10004.436,E2 -10004.436} C_VEL
LIN {X 0,Y 423.494,Z 439.565,A -85,B 0,C 180,E1 -10005.028,E2 -10005.028} C_VEL
LIN {X 0,Y 423.903,Z 426.232,A -85,B 0,C 180,E1 -10005.439,E2 -10005.439} C_VEL
LIN {X 0,Y 424.679,Z 337.02,A -85,B 0,C 180,E1 -10006.888,E2 -10006.888} C_VEL
LIN {X 0,Y 420.637,Z 313.178,A -85,B 0,C 180,E1 -10007.502,E2 -10007.502} C_VEL
LIN {X 0,Y 420.985,Z 305.925,A -85,B 0,C 180,E1 -10008.745,E2 -10008.745} C_VEL
LIN {X 0,Y 422.259,Z 287.874,A -85,B 0,C 180,E1 -10011.992,E2 -10011.992} C_VEL
LIN {X 0,Y 422.977,Z 277.133,A -85,B 0,C 180,E1 -10013.955,E2 -10013.955} C_VEL
LIN {X 0,Y 419.961,Z 262.964,A -85,B 0,C 180,E1 -10016.861,E2 -10016.861} C_VEL
LIN {X 0,Y 418.333,Z 256.091,A -85,B 0,C 180,E1 -10018.367,E2 -10018.367} C_VEL
LIN {X 0,Y 418.214,Z 256.017,A -85,B 0,C 180,E1 -10021.395,E2 -10021.395} C_VEL
LIN {X 0,Y 418.266,Z 255.994,A -85,B 0,C 180,E1 -10024.579,E2 -10024.579} C_VEL
LIN {X 0,Y 418.229,Z 256.009,A -85,B 0,C 180,E1 -10027.833,E2 -10027.833} C_VEL
LIN {X 0,Y 418.223,Z 256.008,A -85,B 0,C 180,E1 -10030.947,E2 -10030.947} C_VEL
LIN {X 0,Y 418.216,Z 256.012,A -85,B 0,C 180,E1 -10033.729,E2 -10033.729} C_VEL
LIN {X 0,Y 418.207,Z 256.011,A -85,B 0,C 180,E1 -10036.448,E2 -10036.448} C_VEL
LIN {X 0,Y 418.221,Z 256.005,A -85,B 0,C 180,E1 -10039.129,E2 -10039.129} C_VEL
LIN {X 0,Y 418.229,Z 256.01,A -85,B 0,C 180,E1 -10042.165,E2 -10042.165} C_VEL
LIN {X 0,Y 418.263,Z 255.993,A -85,B 0,C 180,E1 -10045.419,E2 -10045.419} C_VEL
LIN {X 0,Y 418.213,Z 256.01,A -85,B 0,C 180,E1 -10048.603,E2 -10048.603} C_VEL
LIN {X 0,Y 418.29,Z 255.998,A -85,B 0,C 180,E1 -10051.936,E2 -10051.936} C_VEL
LIN {X 0,Y 418.285,Z 256.001,A -85,B 0,C 180,E1 -10055.162,E2 -10055.162} C_VEL
LIN {X 0,Y 418.229,Z 256.013,A -85,B 0,C 180,E1 -10058.303,E2 -10058.303} C_VEL
LIN {X 0,Y 418.278,Z 256.005,A -85,B 0,C 180,E1 -10061.382,E2 -10061.382} C_VEL
LIN {X 0,Y 418.297,Z 256.003,A -85,B 0,C 180,E1 -10064.405,E2 -10064.405} C_VEL
LIN {X 0,Y 418.35,Z 255.996,A -85,B 0,C 180,E1 -10067.385,E2 -10067.385} C_VEL
LIN {X 0,Y 418.335,Z 255.993,A -85,B 0,C 180,E1 -10070.328,E2 -10070.328} C_VEL
LIN {X 0,Y 418.486,Z 255.979,A -85,B 0,C 180,E1 -10073.249,E2 -10073.249} C_VEL
LIN {X 0,Y 418.334,Z 255.99,A -85,B 0,C 180,E1 -10075.181,E2 -10075.181} C_VEL
LIN {X 0,Y 418.538,Z 255.974,A -85,B 0,C 180,E1 -10078.075,E2 -10078.075} C_VEL
LIN {X 0,Y 418.665,Z 255.956,A -85,B 0,C 180,E1 -10080,E2 -10080} C_VEL
LIN {X 0,Y 418.504,Z 255.978,A -85,B 0,C 180,E1 -10082.887,E2 -10082.887} C_VEL
LIN {X 0,Y 418.487,Z 255.979,A -85,B 0,C 180,E1 -10086.751,E2 -10086.751} C_VEL
LIN {X 0,Y 418.393,Z 255.992,A -85,B 0,C 180,E1 -10088.695,E2 -10088.695} C_VEL
LIN {X 0,Y 418.308,Z 255.994,A -85,B 0,C 180,E1 -10091.631,E2 -10091.631} C_VEL
LIN {X 0,Y 418.296,Z 256.002,A -85,B 0,C 180,E1 -10094.597,E2 -10094.597} C_VEL
LIN {X 0,Y 418.281,Z 256.004,A -85,B 0,C 180,E1 -10097.604,E2 -10097.604} C_VEL
LIN {X 0,Y 418.243,Z 256.007,A -85,B 0,C 180,E1 -10100.663,E2 -10100.663} C_VEL
LIN {X 0,Y 418.282,Z 256.008,A -85,B 0,C 180,E1 -10103.781,E2 -10103.781} C_VEL
LIN {X 0,Y 418.304,Z 256.002,A -85,B 0,C 180,E1 -10107.071,E2 -10107.071} C_VEL
LIN {X 0,Y 418.255,Z 255.991,A -85,B 0,C 180,E1 -10110.271,E2 -10110.271} C_VEL
LIN {X 0,Y 418.243,Z 256.013,A -85,B 0,C 180,E1 -10113.677,E2 -10113.677} C_VEL
LIN {X 0,Y 418.24,Z 255.996,A -85,B 0,C 180,E1 -10117.224,E2 -10117.224} C_VEL
LIN {X 0,Y 418.25,Z 256.015,A -85,B 0,C 180,E1 -10119.682,E2 -10119.682} C_VEL
LIN {X 0,Y 418.225,Z 256.004,A -85,B 0,C 180,E1 -10122.322,E2 -10122.322} C_VEL
LIN {X 0,Y 418.232,Z 256.012,A -85,B 0,C 180,E1 -10125.109,E2 -10125.109} C_VEL
LIN {X 0,Y 418.236,Z 255.978,A -85,B 0,C 180,E1 -10127.767,E2 -10127.767} C_VEL
LIN {X 0,Y 418.254,Z 256.008,A -85,B 0,C 180,E1 -10130.619,E2 -10130.619} C_VEL
LIN {X 0,Y 418.24,Z 255.989,A -85,B 0,C 180,E1 -10133.976,E2 -10133.976} C_VEL
LIN {X 0,Y 418.255,Z 256.004,A -85,B 0,C 180,E1 -10137.157,E2 -10137.157} C_VEL
LIN {X 0,Y 418.293,Z 256.181,A -85,B 0,C 180,E1 -10140.254,E2 -10140.254} C_VEL
LIN {X 0,Y 421.869,Z 270.525,A -85,B 0,C 180,E1 -10143.027,E2 -10143.027} C_VEL
LIN {X 0,Y 423.83,Z 279.8,A -85,B 0,C 180,E1 -10144.724,E2 -10144.724} C_VEL
LIN {X 0,Y 422.271,Z 297.747,A -85,B 0,C 180,E1 -10147.6,E2 -10147.6} C_VEL
LIN {X 0,Y 425.639,Z 319.047,A -85,B 0,C 180,E1 -10148.185,E2 -10148.185} C_VEL
LIN {X 0,Y 423.861,Z 432.434,A -85,B 0,C 180,E1 -10150.224,E2 -10150.224} C_VEL
LIN {X 0,Y 423.327,Z 446.653,A -85,B 0,C 180,E1 -10150.671,E2 -10150.671} C_VEL
LIN {X 0,Y 422.672,Z 461.006,A -85,B 0,C 180,E1 -10151.333,E2 -10151.333} C_VEL
LIN {X 0,Y 421.884,Z 474.798,A -85,B 0,C 180,E1 -10152.187,E2 -10152.187} C_VEL
LIN {X 0,Y 420.961,Z 486.91,A -85,B 0,C 180,E1 -10153.138,E2 -10153.138} C_VEL
LIN {X 0,Y 420.031,Z 499.241,A -85,B 0,C 180,E1 -10154.348,E2 -10154.348} C_VEL
LIN {X 0,Y 419.379,Z 508.495,A -85,B 0,C 180,E1 -10155.442,E2 -10155.442} C_VEL
LIN {X 0,Y 418.733,Z 518.985,A -85,B 0,C 180,E1 -10156.944,E2 -10156.944} C_VEL
LIN {X 0,Y 418.062,Z 528.479,A -85,B 0,C 180,E1 -10158.608,E2 -10158.608} C_VEL
LIN {X 0,Y 417.588,Z 536.333,A -85,B 0,C 180,E1 -10160.311,E2 -10160.311} C_VEL
LIN {X 0,Y 417.31,Z 541.77,A -85,B 0,C 180,E1 -10161.77,E2 -10161.77} C_VEL
LIN {X 0,Y 417.168,Z 546.196,A -85,B 0,C 180,E1 -10163.228,E2 -10163.228} C_VEL
LIN {X 0,Y 417.068,Z 550.633,A -85,B 0,C 180,E1 -10165.167,E2 -10165.167} C_VEL
LIN {X 0,Y 417.024,Z 553.556,A -85,B 0,C 180,E1 -10167.102,E2 -10167.102} C_VEL
LIN {X 0,Y 417.053,Z 554.477,A -85,B 0,C 180,E1 -10168.069,E2 -10168.069} C_VEL
LIN {X 0,Y 417.002,Z 555.255,A -85,B 0,C 180,E1 -10170,E2 -10170} C_VEL
LIN {X 0,Y 417.053,Z 554.616,A -85,B 0,C 180,E1 -10171.931,E2 -10171.931} C_VEL
LIN {X 0,Y 417.001,Z 552.538,A -85,B 0,C 180,E1 -10173.865,E2 -10173.865} C_VEL
LIN {X 0,Y 417.093,Z 548.998,A -85,B 0,C 180,E1 -10175.802,E2 -10175.802} C_VEL
LIN {X 0,Y 417.261,Z 543.896,A -85,B 0,C 180,E1 -10177.744,E2 -10177.744} C_VEL
